LIN {X 0,Y 172.926,Z 518.236,A -85,B 0,C 180,E1 -23636.725,E2 -23636.725} C_VEL
LIN {X 0,Y 167.935,Z 527.248,A -85,B 0,C 180,E1 -23640.546,E2 -23640.546} C_VEL
LIN {X 0,Y 163.837,Z 534.508,A -85,B 0,C 180,E1 -23644.598,E2 -23644.598} C_VEL
LIN {X 0,Y 160.993,Z 539.589,A -85,B 0,C 180,E1 -23648.219,E2 -23648.219} C_VEL
LIN {X 0,Y 157.873,Z 544.852,A -85,B 0,C 180,E1 -23653.181,E2 -23653.181} C_VEL
LIN {X 0,Y 156.336,Z 547.79,A -85,B 0,C 180,E1 -23657.011,E2 -23657.011} C_VEL
LIN {X 0,Y 155.16,Z 550.483,A -85,B 0,C 180,E1 -23662.19,E2 -23662.19} C_VEL
LIN {X 0,Y 154.667,Z 551.827,A -85,B 0,C 180,E1 -23667.396,E2 -23667.396} C_VEL
LIN {X 0,Y 154.657,Z 551.936,A -85,B 0,C 180,E1 -23671.301,E2 -23671.301} C_VEL
LIN {X 0,Y 154.801,Z 551.368,A -85,B 0,C 180,E1 -23675.21,E2 -23675.21} C_VEL
LIN {X 0,Y 155.156,Z 550.552,A -85,B 0,C 180,E1 -23677.81,E2 -23677.81} C_VEL
LIN {X 0,Y 156.317,Z 547.899,A -85,B 0,C 180,E1 -23682.991,E2 -23682.991} C_VEL
LIN {X 0,Y 158.464,Z 543.823,A -85,B 0,C 180,E1 -23688.087,E2 -23688.087} C_VEL
LIN {X 0,Y 161.821,Z 538.19,A -85,B 0,C 180,E1 -23693.009,E2 -23693.009} C_VEL
LIN {X 0,Y 164.996,Z 532.618,A -85,B 0,C 180,E1 -23696.715,E2 -23696.715} C_VEL
LIN {X 0,Y 169.249,Z 525.15,A -85,B 0,C 180,E1 -23700.576,E2 -23700.576} C_VEL
LIN {X 0,Y 173.636,Z 517.128,A -85,B 0,C 180,E1 -23703.817,E2 -23703.817} C_VEL
LIN {X 0,Y 178.54,Z 507.453,A -85,B 0,C 180,E1 -23706.892,E2 -23706.892} C_VEL
LIN {X 0,Y 182.704,Z 498.37,A -85,B 0,C 180,E1 -23709.202,E2 -23709.202} C_VEL
LIN {X 0,Y 183.404,Z 491.819,A -85,B 0,C 180,E1 -23711.15,E2 -23711.15} C_VEL
LIN {X 0,Y 183.287,Z 481.855,A -85,B 0,C 180,E1 -23714.112,E2 -23714.112} C_VEL
LIN {X 0,Y 182.291,Z 472.749,A -85,B 0,C 180,E1 -23716.817,E2 -23716.817} C_VEL
LIN {X 0,Y 180.315,Z 464.485,A -85,B 0,C 180,E1 -23719.466,E2 -23719.466} C_VEL
LIN {X 0,Y 177.999,Z 458.041,A -85,B 0,C 180,E1 -23721.775,E2 -23721.775} C_VEL
LIN {X 0,Y 174.457,Z 449.919,A -85,B 0,C 180,E1 -23724.966,E2 -23724.966} C_VEL
LIN {X 0,Y 171.581,Z 444.63,A -85,B 0,C 180,E1 -23727.392,E2 -23727.392} C_VEL
LIN {X 0,Y 169.45,Z 440.565,A -85,B 0,C 180,E1 -23729.308,E2 -23729.308} C_VEL
LIN {X 0,Y 166.805,Z 436.801,A -85,B 0,C 180,E1 -23731.534,E2 -23731.534} C_VEL
LIN {X 0,Y 165.956,Z 434.977,A -85,B 0,C 180,E1 -23732.407,E2 -23732.407} C_VEL
LIN {X 0,Y 163.2,Z 432.01,A -85,B 0,C 180,E1 -23734.833,E2 -23734.833} C_VEL
LIN {X 0,Y 161.872,Z 429.259,A -85,B 0,C 180,E1 -23736.321,E2 -23736.321} C_VEL
LIN {X 0,Y 159.325,Z 427.59,A -85,B 0,C 180,E1 -23738.828,E2 -23738.828} C_VEL
LIN {X 0,Y 157.743,Z 424.933,A -85,B 0,C 180,E1 -23740.804,E2 -23740.804} C_VEL
LIN {X 0,Y 157.405,Z 423.504,A -85,B 0,C 180,E1 -23741.446,E2 -23741.446} C_VEL
LIN {X 0,Y 157.557,Z 423.483,A -85,B 0,C 180,E1 -23747.113,E2 -23747.113} C_VEL
LIN {X 0,Y 157.775,Z 423.457,A -85,B 0,C 180,E1 -23749.736,E2 -23749.736} C_VEL
LIN {X 0,Y 157.827,Z 423.452,A -85,B 0,C 180,E1 -23752.323,E2 -23752.323} C_VEL
LIN {X 0,Y 158.26,Z 423.396,A -85,B 0,C 180,E1 -23760,E2 -23760} C_VEL
LIN {X 0,Y 157.827,Z 423.449,A -85,B 0,C 180,E1 -23767.677,E2 -23767.677} C_VEL
LIN {X 0,Y 157.708,Z 423.466,A -85,B 0,C 180,E1 -23771.362,E2 -23771.362} C_VEL
LIN {X 0,Y 157.481,Z 423.493,A -85,B 0,C 180,E1 -23775.531,E2 -23775.531} C_VEL
LIN {X 0,Y 157.471,Z 423.801,A -85,B 0,C 180,E1 -23778.604,E2 -23778.604} C_VEL
LIN {X 0,Y 158.285,Z 426.09,A -85,B 0,C 180,E1 -23779.816,E2 -23779.816} C_VEL
LIN {X 0,Y 160.246,Z 428.772,A -85,B 0,C 180,E1 -23782.057,E2 -23782.057} C_VEL
LIN {X 0,Y 162.347,Z 430.594,A -85,B 0,C 180,E1 -23784.114,E2 -23784.114} C_VEL
LIN {X 0,Y 164.079,Z 434.137,A -85,B 0,C 180,E1 -23785.974,E2 -23785.974} C_VEL
LIN {X 0,Y 166.374,Z 436.806,A -85,B 0,C 180,E1 -23787.969,E2 -23787.969} C_VEL
LIN {X 0,Y 168.403,Z 440.705,A -85,B 0,C 180,E1 -23789.88,E2 -23789.88} C_VEL
LIN {X 0,Y 169.659,Z 442.431,A -85,B 0,C 180,E1 -23790.887,E2 -23790.887} C_VEL
LIN {X 0,Y 172.027,Z 446.791,A -85,B 0,C 180,E1 -23792.947,E2 -23792.947} C_VEL
LIN {X 0,Y 175.71,Z 454.541,A -85,B 0,C 180,E1 -23796.154,E2 -23796.154} C_VEL
LIN {X 0,Y 178.774,Z 462.124,A -85,B 0,C 180,E1 -23798.976,E2 -23798.976} C_VEL
LIN {X 0,Y 181.187,Z 470.196,A -85,B 0,C 180,E1 -23801.677,E2 -23801.677} C_VEL
LIN {X 0,Y 182.199,Z 476.723,A -85,B 0,C 180,E1 -23803.59,E2 -23803.59} C_VEL
LIN {X 0,Y 182.759,Z 485.981,A -85,B 0,C 180,E1 -23806.196,E2 -23806.196} C_VEL
LIN {X 0,Y 182.442,Z 495.967,A -85,B 0,C 180,E1 -23809.09,E2 -23809.09} C_VEL
LIN {X 0,Y 181.954,Z 500.895,A -85,B 0,C 180,E1 -23810.579,E2 -23810.579} C_VEL
LIN {X 0,Y 181.533,Z 502.814,A -85,B 0,C 180,E1 -23811.119,E2 -23811.119} C_VEL
LIN {X 0,Y 176.391,Z 513.568,A -85,B 0,C 180,E1 -23814.006,E2 -23814.006} C_VEL
LIN {X 0,Y 171.669,Z 522.688,A -85,B 0,C 180,E1 -23817.149,E2 -23817.149} C_VEL
LIN {X 0,Y 166.779,Z 531.405,A -85,B 0,C 180,E1 -23821.013,E2 -23821.013} C_VEL
LIN {X 0,Y 162.662,Z 538.52,A -85,B 0,C 180,E1 -23825.139,E2 -23825.139} C_VEL
LIN {X 0,Y 159.677,Z 544.066,A -85,B 0,C 180,E1 -23829.383,E2 -23829.383} C_VEL
LIN {X 0,Y 156.925,Z 548.946,A -85,B 0,C 180,E1 -23834.412,E2 -23834.412} C_VEL
LIN {X 0,Y 155.389,Z 552.34,A -85,B 0,C 180,E1 -23839.577,E2 -23839.577} C_VEL
LIN {X 0,Y 154.695,Z 554.346,A -85,B 0,C 180,E1 -23844.786,E2 -23844.786} C_VEL
LIN {X 0,Y 154.684,Z 555.005,A -85,B 0,C 180,E1 -23850,E2 -23850} C_VEL
LIN {X 0,Y 154.695,Z 554.325,A -85,B 0,C 180,E1 -23855.213,E2 -23855.213} C_VEL
LIN {X 0,Y 155.39,Z 552.301,A -85,B 0,C 180,E1 -23860.423,E2 -23860.423} C_VEL
LIN {X 0,Y 156.92,Z 548.885,A -85,B 0,C 180,E1 -23865.588,E2 -23865.588} C_VEL
LIN {X 0,Y 159.688,Z 543.979,A -85,B 0,C 180,E1 -23870.615,E2 -23870.615} C_VEL
LIN {X 0,Y 162.854,Z 538.174,A -85,B 0,C 180,E1 -23875.007,E2 -23875.007} C_VEL
LIN {X 0,Y 166.773,Z 531.27,A -85,B 0,C 180,E1 -23878.988,E2 -23878.988} C_VEL
LIN {X 0,Y 171.692,Z 522.522,A -85,B 0,C 180,E1 -23882.845,E2 -23882.845} C_VEL
LIN {X 0,Y 176.409,Z 513.368,A -85,B 0,C 180,E1 -23885.989,E2 -23885.989} C_VEL
LIN {X 0,Y 178.015,Z 510.091,A -85,B 0,C 180,E1 -23886.936,E2 -23886.936} C_VEL
LIN {X 0,Y 178.978,Z 507.362,A -85,B 0,C 180,E1 -23887.774,E2 -23887.774} C_VEL
LIN {X 0,Y 179.272,Z 503.359,A -85,B 0,C 180,E1 -23889.176,E2 -23889.176} C_VEL
LIN {X 0,Y 178.699,Z 499.6,A -85,B 0,C 180,E1 -23890.654,E2 -23890.654} C_VEL
LIN {X 0,Y 177.025,Z 491.821,A -85,B 0,C 180,E1 -23893.689,E2 -23893.689} C_VEL
LIN {X 0,Y 176.838,Z 488.942,A -85,B 0,C 180,E1 -23894.631,E2 -23894.631} C_VEL
LIN {X 0,Y 176.635,Z 479.607,A -85,B 0,C 180,E1 -23897.437,E2 -23897.437} C_VEL
LIN {X 0,Y 175.522,Z 472.284,A -85,B 0,C 180,E1 -23899.778,E2 -23899.778} C_VEL
LIN {X 0,Y 173.933,Z 466.481,A -85,B 0,C 180,E1 -23901.855,E2 -23901.855} C_VEL
LIN {X 0,Y 171.092,Z 458.845,A -85,B 0,C 180,E1 -23904.895,E2 -23904.895} C_VEL
LIN {X 0,Y 168.211,Z 452.209,A -85,B 0,C 180,E1 -23907.812,E2 -23907.812} C_VEL
LIN {X 0,Y 166.109,Z 447.895,A -85,B 0,C 180,E1 -23909.927,E2 -23909.927} C_VEL
LIN {X 0,Y 163.64,Z 443.734,A -85,B 0,C 180,E1 -23912.33,E2 -23912.33} C_VEL
LIN {X 0,Y 163.002,Z 442.254,A -85,B 0,C 180,E1 -23913.082,E2 -23913.082} C_VEL
LIN {X 0,Y 160.807,Z 439.375,A -85,B 0,C 180,E1 -23915.242,E2 -23915.242} C_VEL
LIN {X 0,Y 159.571,Z 436.565,A -85,B 0,C 180,E1 -23916.819,E2 -23916.819} C_VEL
LIN {X 0,Y 156.742,Z 433.546,A -85,B 0,C 180,E1 -23920.017,E2 -23920.017} C_VEL
LIN {X 0,Y 155.337,Z 430.302,A -85,B 0,C 180,E1 -23922.218,E2 -23922.218} C_VEL
LIN {X 0,Y 152.287,Z 428.264,A -85,B 0,C 180,E1 -23926.81,E2 -23926.81} C_VEL
LIN {X 0,Y 150.954,Z 425.405,A -85,B 0,C 180,E1 -23930.03,E2 -23930.03} C_VEL
LIN {X 0,Y 150.722,Z 424.337,A -85,B 0,C 180,E1 -23930.946,E2 -23930.946} C_VEL
LIN {X 0,Y 150.903,Z 424.313,A -85,B 0,C 180,E1 -23937.331,E2 -23937.331} C_VEL
LIN {X 0,Y 151.221,Z 424.272,A -85,B 0,C 180,E1 -23940,E2 -23940} C_VEL
LIN {X 0,Y 150.764,Z 424.33,A -85,B 0,C 180,E1 -23948.039,E2 -23948.039} C_VEL
LIN {X 0,Y 150.746,Z 424.431,A -85,B 0,C 180,E1 -23949.391,E2 -23949.391} C_VEL
LIN {X 0,Y 151.619,Z 427.253,A -85,B 0,C 180,E1 -23952.009,E2 -23952.009} C_VEL
LIN {X 0,Y 153.548,Z 429.386,A -85,B 0,C 180,E1 -23955.599,E2 -23955.599} C_VEL
LIN {X 0,Y 155.496,Z 430.531,A -85,B 0,C 180,E1 -23958.274,E2 -23958.274} C_VEL
LIN {X 0,Y 156.695,Z 433.412,A -85,B 0,C 180,E1 -23960.169,E2 -23960.169} C_VEL
LIN {X 0,Y 159.006,Z 435.579,A -85,B 0,C 180,E1 -23962.795,E2 -23962.795} C_VEL
LIN {X 0,Y 159.683,Z 436.232,A -85,B 0,C 180,E1 -23963.514,E2 -23963.514} C_VEL
LIN {X 0,Y 161.638,Z 439.756,A -85,B 0,C 180,E1 -23965.773,E2 -23965.773} C_VEL
LIN {X 0,Y 163.321,Z 441.724,A -85,B 0,C 180,E1 -23967.381,E2 -23967.381} C_VEL
LIN {X 0,Y 166.904,Z 448.442,A -85,B 0,C 180,E1 -23971.053,E2 -23971.053} C_VEL
LIN {X 0,Y 168.703,Z 451.832,A -85,B 0,C 180,E1 -23972.791,E2 -23972.791} C_VEL
LIN {X 0,Y 171.618,Z 458.27,A -85,B 0,C 180,E1 -23975.701,E2 -23975.701} C_VEL
LIN {X 0,Y 174.36,Z 465.65,A -85,B 0,C 180,E1 -23978.665,E2 -23978.665} C_VEL
LIN {X 0,Y 176.184,Z 472.574,A -85,B 0,C 180,E1 -23981.161,E2 -23981.161} C_VEL
LIN {X 0,Y 177.218,Z 479.908,A -85,B 0,C 180,E1 -23983.566,E2 -23983.566} C_VEL
LIN {X 0,Y 177.528,Z 489.397,A -85,B 0,C 180,E1 -23986.532,E2 -23986.532} C_VEL
LIN {X 0,Y 176.984,Z 497.901,A -85,B 0,C 180,E1 -23989.268,E2 -23989.268} C_VEL
LIN {X 0,Y 176.815,Z 499.083,A -85,B 0,C 180,E1 -23989.638,E2 -23989.638} C_VEL
LIN {X 0,Y 172.036,Z 508.857,A -85,B 0,C 180,E1 -23992.21,E2 -23992.21} C_VEL
LIN {X 0,Y 167.013,Z 518.308,A -85,B 0,C 180,E1 -23995.383,E2 -23995.383} C_VEL
LIN {X 0,Y 161.766,Z 527.319,A -85,B 0,C 180,E1 -23999.304,E2 -23999.304} C_VEL
LIN {X 0,Y 157.381,Z 534.579,A -85,B 0,C 180,E1 -24003.477,E2 -24003.477} C_VEL
LIN {X 0,Y 154.393,Z 539.66,A -85,B 0,C 180,E1 -24007.237,E2 -24007.237} C_VEL
LIN {X 0,Y 151.045,Z 544.923,A -85,B 0,C 180,E1 -24012.396,E2 -24012.396} C_VEL
LIN {X 0,Y 149.41,Z 547.859,A -85,B 0,C 180,E1 -24016.397,E2 -24016.397} C_VEL
LIN {X 0,Y 148.102,Z 550.552,A -85,B 0,C 180,E1 -24021.816,E2 -24021.816} C_VEL
LIN {X 0,Y 147.572,Z 551.896,A -85,B 0,C 180,E1 -24027.271,E2 -24027.271} C_VEL
LIN {X 0,Y 147.597,Z 552.049,A -85,B 0,C 180,E1 -24030.614,E2 -24030.614} C_VEL
LIN {X 0,Y 147.727,Z 551.437,A -85,B 0,C 180,E1 -24035.46,E2 -24035.46} C_VEL
LIN {X 0,Y 148.604,Z 549.466,A -85,B 0,C 180,E1 -24040.905,E2 -24040.905} C_VEL
LIN {X 0,Y 150.419,Z 546.114,A -85,B 0,C 180,E1 -24046.281,E2 -24046.281} C_VEL
LIN {X 0,Y 153.413,Z 541.278,A -85,B 0,C 180,E1 -24051.499,E2 -24051.499} C_VEL
LIN {X 0,Y 157.396,Z 534.805,A -85,B 0,C 180,E1 -24056.521,E2 -24056.521} C_VEL
LIN {X 0,Y 161.734,Z 527.596,A -85,B 0,C 180,E1 -24060.703,E2 -24060.703} C_VEL
LIN {X 0,Y 166.938,Z 518.674,A -85,B 0,C 180,E1 -24064.635,E2 -24064.635} C_VEL
LIN {X 0,Y 172.006,Z 509.298,A -85,B 0,C 180,E1 -24067.799,E2 -24067.799} C_VEL
LIN {X 0,Y 176.72,Z 499.621,A -85,B 0,C 180,E1 -24070.386,E2 -24070.386} C_VEL
LIN {X 0,Y 177.522,Z 492.221,A -85,B 0,C 180,E1 -24072.722,E2 -24072.722} C_VEL
LIN {X 0,Y 177.517,Z 482.496,A -85,B 0,C 180,E1 -24075.784,E2 -24075.784} C_VEL
LIN {X 0,Y 176.693,Z 474.887,A -85,B 0,C 180,E1 -24078.223,E2 -24078.223} C_VEL
LIN {X 0,Y 175.181,Z 468.219,A -85,B 0,C 180,E1 -24080.558,E2 -24080.558} C_VEL
LIN {X 0,Y 172.912,Z 461.554,A -85,B 0,C 180,E1 -24083.165,E2 -24083.165} C_VEL
LIN {X 0,Y 170.239,Z 454.885,A -85,B 0,C 180,E1 -24085.986,E2 -24085.986} C_VEL
LIN {X 0,Y 167.733,Z 449.906,A -85,B 0,C 180,E1 -24088.416,E2 -24088.416} C_VEL
LIN {X 0,Y 165.651,Z 445.799,A -85,B 0,C 180,E1 -24090.535,E2 -24090.535} C_VEL
LIN {X 0,Y 163.358,Z 441.764,A -85,B 0,C 180,E1 -24092.886,E2 -24092.886} C_VEL
LIN {X 0,Y 160.147,Z 437.275,A -85,B 0,C 180,E1 -24096.222,E2 -24096.222} C_VEL
LIN {X 0,Y 159.511,Z 435.836,A -85,B 0,C 180,E1 -24097.067,E2 -24097.067} C_VEL
LIN {X 0,Y 157.043,Z 433.825,A -85,B 0,C 180,E1 -24099.796,E2 -24099.796} C_VEL
LIN {X 0,Y 155.502,Z 430.56,A -85,B 0,C 180,E1 -24102.152,E2 -24102.152} C_VEL
LIN {X 0,Y 152.111,Z 427.998,A -85,B 0,C 180,E1 -24107.546,E2 -24107.546} C_VEL
LIN {X 0,Y 150.805,Z 424.729,A -85,B 0,C 180,E1 -24111.204,E2 -24111.204} C_VEL
LIN {X 0,Y 150.749,Z 424.33,A -85,B 0,C 180,E1 -24111.623,E2 -24111.623} C_VEL
LIN {X 0,Y 151.221,Z 424.273,A -85,B 0,C 180,E1 -24120,E2 -24120} C_VEL
LIN {X 0,Y 150.739,Z 424.365,A -85,B 0,C 180,E1 -24128.378,E2 -24128.378} C_VEL
LIN {X 0,Y 151.542,Z 426.956,A -85,B 0,C 180,E1 -24130.996,E2 -24130.996} C_VEL
LIN {X 0,Y 153.348,Z 429.262,A -85,B 0,C 180,E1 -24134.6,E2 -24134.6} C_VEL
LIN {X 0,Y 155.559,Z 430.611,A -85,B 0,C 180,E1 -24137.755,E2 -24137.755} C_VEL
LIN {X 0,Y 157.293,Z 434.31,A -85,B 0,C 180,E1 -24140.38,E2 -24140.38} C_VEL
LIN {X 0,Y 159.896,Z 437.055,A -85,B 0,C 180,E1 -24143.302,E2 -24143.302} C_VEL
LIN {X 0,Y 161.729,Z 440.76,A -85,B 0,C 180,E1 -24145.498,E2 -24145.498} C_VEL
LIN {X 0,Y 163.385,Z 442.899,A -85,B 0,C 180,E1 -24147.109,E2 -24147.109} C_VEL
LIN {X 0,Y 165.56,Z 447.084,A -85,B 0,C 180,E1 -24149.395,E2 -24149.395} C_VEL
LIN {X 0,Y 166.06,Z 447.7,A -85,B 0,C 180,E1 -24149.82,E2 -24149.82} C_VEL
LIN {X 0,Y 168.931,Z 453.785,A -85,B 0,C 180,E1 -24152.74,E2 -24152.74} C_VEL
LIN {X 0,Y 172.407,Z 461.832,A -85,B 0,C 180,E1 -24156.233,E2 -24156.233} C_VEL
LIN {X 0,Y 175.431,Z 471.484,A -85,B 0,C 180,E1 -24159.865,E2 -24159.865} C_VEL
LIN {X 0,Y 176.511,Z 477.442,A -85,B 0,C 180,E1 -24161.829,E2 -24161.829} C_VEL
LIN {X 0,Y 176.965,Z 486.961,A -85,B 0,C 180,E1 -24164.692,E2 -24164.692} C_VEL
LIN {X 0,Y 176.609,Z 495.895,A -85,B 0,C 180,E1 -24167.429,E2 -24167.429} C_VEL
LIN {X 0,Y 175.69,Z 503.255,A -85,B 0,C 180,E1 -24169.76,E2 -24169.76} C_VEL
LIN {X 0,Y 171.568,Z 511.821,A -85,B 0,C 180,E1 -24172.088,E2 -24172.088} C_VEL
LIN {X 0,Y 166.469,Z 521.245,A -85,B 0,C 180,E1 -24175.253,E2 -24175.253} C_VEL
LIN {X 0,Y 161.277,Z 530.22,A -85,B 0,C 180,E1 -24179.2,E2 -24179.2} C_VEL
LIN {X 0,Y 156.849,Z 537.475,A -85,B 0,C 180,E1 -24183.38,E2 -24183.38} C_VEL
LIN {X 0,Y 152.987,Z 543.998,A -85,B 0,C 180,E1 -24188.438,E2 -24188.438} C_VEL
LIN {X 0,Y 150.057,Z 548.877,A -85,B 0,C 180,E1 -24193.679,E2 -24193.679} C_VEL
LIN {X 0,Y 148.374,Z 552.271,A -85,B 0,C 180,E1 -24199.078,E2 -24199.078} C_VEL
LIN {X 0,Y 147.623,Z 554.277,A -85,B 0,C 180,E1 -24204.536,E2 -24204.536} C_VEL
LIN {X 0,Y 147.588,Z 554.936,A -85,B 0,C 180,E1 -24210,E2 -24210} C_VEL
LIN {X 0,Y 147.623,Z 554.255,A -85,B 0,C 180,E1 -24215.463,E2 -24215.463} C_VEL
LIN {X 0,Y 148.374,Z 552.231,A -85,B 0,C 180,E1 -24220.921,E2 -24220.921} C_VEL
LIN {X 0,Y 150.053,Z 548.815,A -85,B 0,C 180,E1 -24226.321,E2 -24226.321} C_VEL
LIN {X 0,Y 153.002,Z 543.908,A -85,B 0,C 180,E1 -24231.56,E2 -24231.56} C_VEL
LIN {X 0,Y 156.143,Z 538.54,A -85,B 0,C 180,E1 -24235.816,E2 -24235.816} C_VEL
LIN {X 0,Y 160.574,Z 531.199,A -85,B 0,C 180,E1 -24240.22,E2 -24240.22} C_VEL
LIN {X 0,Y 165.74,Z 522.451,A -85,B 0,C 180,E1 -24244.184,E2 -24244.184} C_VEL
LIN {X 0,Y 170.696,Z 513.296,A -85,B 0,C 180,E1 -24247.394,E2 -24247.394} C_VEL
LIN {X 0,Y 175.66,Z 503.055,A -85,B 0,C 180,E1 -24250.228,E2 -24250.228} C_VEL
LIN {X 0,Y 176.704,Z 493.056,A -85,B 0,C 180,E1 -24253.378,E2 -24253.378} C_VEL
LIN {X 0,Y 176.838,Z 488.942,A -85,B 0,C 180,E1 -24254.631,E2 -24254.631} C_VEL
LIN {X 0,Y 176.306,Z 484.941,A -85,B 0,C 180,E1 -24256.029,E2 -24256.029} C_VEL
LIN {X 0,Y 174.873,Z 481.493,A -85,B 0,C 180,E1 -24257.542,E2 -24257.542} C_VEL
LIN {X 0,Y 169.938,Z 473.071,A -85,B 0,C 180,E1 -24261.821,E2 -24261.821} C_VEL
LIN {X 0,Y 169.036,Z 470.649,A -85,B 0,C 180,E1 -24262.874,E2 -24262.874} C_VEL
LIN {X 0,Y 166.521,Z 463.123,A -85,B 0,C 180,E1 -24266.094,E2 -24266.094} C_VEL
LIN {X 0,Y 163.981,Z 456.991,A -85,B 0,C 180,E1 -24269.049,E2 -24269.049} C_VEL
LIN {X 0,Y 162.458,Z 453.39,A -85,B 0,C 180,E1 -24270.878,E2 -24270.878} C_VEL
LIN {X 0,Y 160.342,Z 449.38,A -85,B 0,C 180,E1 -24273.303,E2 -24273.303} C_VEL
LIN {X 0,Y 159.278,Z 447.608,A -85,B 0,C 180,E1 -24274.519,E2 -24274.519} C_VEL
LIN {X 0,Y 157.237,Z 443.663,A -85,B 0,C 180,E1 -24277.151,E2 -24277.151} C_VEL
LIN {X 0,Y 156.533,Z 442.51,A -85,B 0,C 180,E1 -24278.086,E2 -24278.086} C_VEL
LIN {X 0,Y 154.245,Z 439.526,A -85,B 0,C 180,E1 -24281.115,E2 -24281.115} C_VEL
LIN {X 0,Y 153.232,Z 436.998,A -85,B 0,C 180,E1 -24282.999,E2 -24282.999} C_VEL
LIN {X 0,Y 150.601,Z 434.94,A -85,B 0,C 180,E1 -24287.42,E2 -24287.42} C_VEL
LIN {X 0,Y 149.422,Z 432.001,A -85,B 0,C 180,E1 -24290.884,E2 -24290.884} C_VEL
LIN {X 0,Y 149.306,Z 431.322,A -85,B 0,C 180,E1 -24291.491,E2 -24291.491} C_VEL
LIN {X 0,Y 147.774,Z 430.484,A -85,B 0,C 180,E1 -24300,E2 -24300} C_VEL
LIN {X 0,Y 149.308,Z 431.378,A -85,B 0,C 180,E1 -24308.8,E2 -24308.8} C_VEL
LIN {X 0,Y 150.294,Z 434.547,A -85,B 0,C 180,E1 -24312.181,E2 -24312.181} C_VEL
LIN {X 0,Y 152.563,Z 436.717,A -85,B 0,C 180,E1 -24316.389,E2 -24316.389} C_VEL
LIN {X 0,Y 153.357,Z 437.198,A -85,B 0,C 180,E1 -24317.524,E2 -24317.524} C_VEL
LIN {X 0,Y 154.614,Z 440.165,A -85,B 0,C 180,E1 -24319.76,E2 -24319.76} C_VEL
LIN {X 0,Y 157.066,Z 442.636,A -85,B 0,C 180,E1 -24322.789,E2 -24322.789} C_VEL
LIN {X 0,Y 158.902,Z 446.104,A -85,B 0,C 180,E1 -24325.195,E2 -24325.195} C_VEL
LIN {X 0,Y 160.283,Z 448.011,A -85,B 0,C 180,E1 -24326.708,E2 -24326.708} C_VEL
LIN {X 0,Y 164.429,Z 456.285,A -85,B 0,C 180,E1 -24331.501,E2 -24331.501} C_VEL
LIN {X 0,Y 167.452,Z 463.802,A -85,B 0,C 180,E1 -24335.089,E2 -24335.089} C_VEL
LIN {X 0,Y 169.914,Z 471.524,A -85,B 0,C 180,E1 -24338.348,E2 -24338.348} C_VEL
LIN {X 0,Y 171.296,Z 478.694,A -85,B 0,C 180,E1 -24341.03,E2 -24341.03} C_VEL
LIN {X 0,Y 171.774,Z 486.393,A -85,B 0,C 180,E1 -24343.664,E2 -24343.664} C_VEL
LIN {X 0,Y 171.489,Z 494.96,A -85,B 0,C 180,E1 -24346.53,E2 -24346.53} C_VEL
LIN {X 0,Y 170.883,Z 500.342,A -85,B 0,C 180,E1 -24348.379,E2 -24348.379} C_VEL
LIN {X 0,Y 165.553,Z 510.633,A -85,B 0,C 180,E1 -24351.233,E2 -24351.233} C_VEL
LIN {X 0,Y 160.395,Z 519.773,A -85,B 0,C 180,E1 -24354.509,E2 -24354.509} C_VEL
LIN {X 0,Y 154.972,Z 528.503,A -85,B 0,C 180,E1 -24358.565,E2 -24358.565} C_VEL
LIN {X 0,Y 151.012,Z 534.65,A -85,B 0,C 180,E1 -24362.265,E2 -24362.265} C_VEL
LIN {X 0,Y 146.849,Z 541.168,A -85,B 0,C 180,E1 -24367.489,E2 -24367.489} C_VEL
LIN {X 0,Y 143.61,Z 546.053,A -85,B 0,C 180,E1 -24372.925,E2 -24372.925} C_VEL
LIN {X 0,Y 141.638,Z 549.448,A -85,B 0,C 180,E1 -24378.552,E2 -24378.552} C_VEL
LIN {X 0,Y 140.655,Z 551.459,A -85,B 0,C 180,E1 -24384.265,E2 -24384.265} C_VEL
LIN {X 0,Y 140.524,Z 552.141,A -85,B 0,C 180,E1 -24390,E2 -24390} C_VEL
LIN {X 0,Y 140.654,Z 551.505,A -85,B 0,C 180,E1 -24395.736,E2 -24395.736} C_VEL
LIN {X 0,Y 141.626,Z 549.535,A -85,B 0,C 180,E1 -24401.449,E2 -24401.449} C_VEL
LIN {X 0,Y 143.572,Z 546.182,A -85,B 0,C 180,E1 -24407.08,E2 -24407.08} C_VEL
LIN {X 0,Y 146.812,Z 541.346,A -85,B 0,C 180,E1 -24412.518,E2 -24412.518} C_VEL
LIN {X 0,Y 151.013,Z 534.873,A -85,B 0,C 180,E1 -24417.736,E2 -24417.736} C_VEL
LIN {X 0,Y 155.647,Z 527.664,A -85,B 0,C 180,E1 -24422.043,E2 -24422.043} C_VEL
LIN {X 0,Y 161.146,Z 518.741,A -85,B 0,C 180,E1 -24426.07,E2 -24426.07} C_VEL
LIN {X 0,Y 166.447,Z 509.364,A -85,B 0,C 180,E1 -24429.298,E2 -24429.298} C_VEL
LIN {X 0,Y 170.824,Z 500.796,A -85,B 0,C 180,E1 -24431.649,E2 -24431.649} C_VEL
LIN {X 0,Y 171.71,Z 492.378,A -85,B 0,C 180,E1 -24434.51,E2 -24434.51} C_VEL
LIN {X 0,Y 171.821,Z 483.724,A -85,B 0,C 180,E1 -24437.414,E2 -24437.414} C_VEL
LIN {X 0,Y 171.166,Z 477.13,A -85,B 0,C 180,E1 -24439.707,E2 -24439.707} C_VEL
LIN {X 0,Y 169.694,Z 470.441,A -85,B 0,C 180,E1 -24442.271,E2 -24442.271} C_VEL
LIN {X 0,Y 166.768,Z 461.825,A -85,B 0,C 180,E1 -24446.035,E2 -24446.035} C_VEL
LIN {X 0,Y 164.149,Z 455.711,A -85,B 0,C 180,E1 -24449.084,E2 -24449.084} C_VEL
LIN {X 0,Y 162.061,Z 451.341,A -85,B 0,C 180,E1 -24451.508,E2 -24451.508} C_VEL
LIN {X 0,Y 160.059,Z 447.326,A -85,B 0,C 180,E1 -24453.954,E2 -24453.954} C_VEL
LIN {X 0,Y 157.548,Z 443.745,A -85,B 0,C 180,E1 -24456.851,E2 -24456.851} C_VEL
LIN {X 0,Y 157.052,Z 442.433,A -85,B 0,C 180,E1 -24457.643,E2 -24457.643} C_VEL
LIN {X 0,Y 154.75,Z 440.25,A -85,B 0,C 180,E1 -24460.489,E2 -24460.489} C_VEL
LIN {X 0,Y 153.336,Z 437.052,A -85,B 0,C 180,E1 -24463.011,E2 -24463.011} C_VEL
LIN {X 0,Y 150.754,Z 435.125,A -85,B 0,C 180,E1 -24467.412,E2 -24467.412} C_VEL
LIN {X 0,Y 149.474,Z 432.114,A -85,B 0,C 180,E1 -24471.305,E2 -24471.305} C_VEL
LIN {X 0,Y 149.186,Z 431.244,A -85,B 0,C 180,E1 -24472.556,E2 -24472.556} C_VEL
LIN {X 0,Y 148.077,Z 430.62,A -85,B 0,C 180,E1 -24480,E2 -24480} C_VEL
LIN {X 0,Y 149.372,Z 431.501,A -85,B 0,C 180,E1 -24487.944,E2 -24487.944} C_VEL
LIN {X 0,Y 150.738,Z 435.101,A -85,B 0,C 180,E1 -24492.34,E2 -24492.34} C_VEL
LIN {X 0,Y 153.53,Z 437.424,A -85,B 0,C 180,E1 -24497.117,E2 -24497.117} C_VEL
LIN {X 0,Y 155.202,Z 441.021,A -85,B 0,C 180,E1 -24499.958,E2 -24499.958} C_VEL
LIN {X 0,Y 157.232,Z 443.385,A -85,B 0,C 180,E1 -24502.503,E2 -24502.503} C_VEL
LIN {X 0,Y 159.202,Z 447.421,A -85,B 0,C 180,E1 -24505.144,E2 -24505.144} C_VEL
LIN {X 0,Y 160.082,Z 448.427,A -85,B 0,C 180,E1 -24506.042,E2 -24506.042} C_VEL
LIN {X 0,Y 162.035,Z 452.746,A -85,B 0,C 180,E1 -24508.496,E2 -24508.496} C_VEL
LIN {X 0,Y 164.531,Z 457.871,A -85,B 0,C 180,E1 -24511.316,E2 -24511.316} C_VEL
LIN {X 0,Y 167.846,Z 466.528,A -85,B 0,C 180,E1 -24515.306,E2 -24515.306} C_VEL
LIN {X 0,Y 170.378,Z 475.691,A -85,B 0,C 180,E1 -24518.98,E2 -24518.98} C_VEL
LIN {X 0,Y 171.169,Z 481.679,A -85,B 0,C 180,E1 -24521.067,E2 -24521.067} C_VEL
LIN {X 0,Y 171.222,Z 490.355,A -85,B 0,C 180,E1 -24523.859,E2 -24523.859} C_VEL
LIN {X 0,Y 170.5,Z 499.166,A -85,B 0,C 180,E1 -24526.743,E2 -24526.743} C_VEL
LIN {X 0,Y 169.709,Z 504.349,A -85,B 0,C 180,E1 -24528.502,E2 -24528.502} C_VEL
LIN {X 0,Y 165.068,Z 513.435,A -85,B 0,C 180,E1 -24531.097,E2 -24531.097} C_VEL
LIN {X 0,Y 159.846,Z 522.554,A -85,B 0,C 180,E1 -24534.368,E2 -24534.368} C_VEL
LIN {X 0,Y 154.473,Z 531.27,A -85,B 0,C 180,E1 -24538.452,E2 -24538.452} C_VEL
LIN {X 0,Y 150.515,Z 537.407,A -85,B 0,C 180,E1 -24542.164,E2 -24542.164} C_VEL
LIN {X 0,Y 147.291,Z 542.495,A -85,B 0,C 180,E1 -24546.072,E2 -24546.072} C_VEL
LIN {X 0,Y 143.907,Z 547.742,A -85,B 0,C 180,E1 -24551.491,E2 -24551.491} C_VEL
LIN {X 0,Y 142.163,Z 550.684,A -85,B 0,C 180,E1 -24555.689,E2 -24555.689} C_VEL
LIN {X 0,Y 140.844,Z 553.375,A -85,B 0,C 180,E1 -24561.39,E2 -24561.39} C_VEL
LIN {X 0,Y 140.42,Z 554.705,A -85,B 0,C 180,E1 -24567.131,E2 -24567.131} C_VEL
LIN {X 0,Y 140.484,Z 554.867,A -85,B 0,C 180,E1 -24570,E2 -24570} C_VEL
LIN {X 0,Y 140.547,Z 554.186,A -85,B 0,C 180,E1 -24575.739,E2 -24575.739} C_VEL
LIN {X 0,Y 141.382,Z 552.162,A -85,B 0,C 180,E1 -24581.469,E2 -24581.469} C_VEL
LIN {X 0,Y 143.211,Z 548.745,A -85,B 0,C 180,E1 -24587.124,E2 -24587.124} C_VEL
LIN {X 0,Y 146.367,Z 543.838,A -85,B 0,C 180,E1 -24592.59,E2 -24592.59} C_VEL
LIN {X 0,Y 149.484,Z 538.884,A -85,B 0,C 180,E1 -24596.711,E2 -24596.711} C_VEL
LIN {X 0,Y 153.753,Z 532.246,A -85,B 0,C 180,E1 -24600.946,E2 -24600.946} C_VEL
LIN {X 0,Y 159.073,Z 523.736,A -85,B 0,C 180,E1 -24605.054,E2 -24605.054} C_VEL
LIN {X 0,Y 164.185,Z 514.854,A -85,B 0,C 180,E1 -24608.365,E2 -24608.365} C_VEL
LIN {X 0,Y 168.863,Z 506.049,A -85,B 0,C 180,E1 -24610.958,E2 -24610.958} C_VEL
LIN {X 0,Y 169.684,Z 504.094,A -85,B 0,C 180,E1 -24611.505,E2 -24611.505} C_VEL
LIN {X 0,Y 170.883,Z 494.42,A -85,B 0,C 180,E1 -24614.742,E2 -24614.742} C_VEL
LIN {X 0,Y 171.196,Z 485.454,A -85,B 0,C 180,E1 -24617.641,E2 -24617.641} C_VEL
LIN {X 0,Y 170.881,Z 479.361,A -85,B 0,C 180,E1 -24619.627,E2 -24619.627} C_VEL
LIN {X 0,Y 169.776,Z 473.177,A -85,B 0,C 180,E1 -24621.861,E2 -24621.861} C_VEL
LIN {X 0,Y 169.036,Z 470.649,A -85,B 0,C 180,E1 -24622.874,E2 -24622.874} C_VEL
LIN {X 0,Y 167.515,Z 467.436,A -85,B 0,C 180,E1 -24624.473,E2 -24624.473} C_VEL
LIN {X 0,Y 165.379,Z 465.053,A -85,B 0,C 180,E1 -24626.195,E2 -24626.195} C_VEL
LIN {X 0,Y 159.311,Z 459.832,A -85,B 0,C 180,E1 -24631.121,E2 -24631.121} C_VEL
LIN {X 0,Y 158.193,Z 458.108,A -85,B 0,C 180,E1 -24632.37,E2 -24632.37} C_VEL
LIN {X 0,Y 156.551,Z 454.204,A -85,B 0,C 180,E1 -24634.756,E2 -24634.756} C_VEL
LIN {X 0,Y 154.691,Z 450.898,A -85,B 0,C 180,E1 -24637.283,E2 -24637.283} C_VEL
LIN {X 0,Y 153.953,Z 448.998,A -85,B 0,C 180,E1 -24638.58,E2 -24638.58} C_VEL
LIN {X 0,Y 151.711,Z 445.764,A -85,B 0,C 180,E1 -24641.953,E2 -24641.953} C_VEL
LIN {X 0,Y 151.079,Z 443.746,A -85,B 0,C 180,E1 -24643.446,E2 -24643.446} C_VEL
LIN {X 0,Y 148.68,Z 441.662,A -85,B 0,C 180,E1 -24647.892,E2 -24647.892} C_VEL
LIN {X 0,Y 147.667,Z 438.63,A -85,B 0,C 180,E1 -24651.594,E2 -24651.594} C_VEL
LIN {X 0,Y 147.463,Z 438.141,A -85,B 0,C 180,E1 -24652.469,E2 -24652.469} C_VEL
LIN {X 0,Y 146.312,Z 437.42,A -85,B 0,C 180,E1 -24660,E2 -24660} C_VEL
LIN {X 0,Y 147.595,Z 438.404,A -85,B 0,C 180,E1 -24668.385,E2 -24668.385} C_VEL
LIN {X 0,Y 148.41,Z 441.314,A -85,B 0,C 180,E1 -24671.784,E2 -24671.784} C_VEL
LIN {X 0,Y 150.848,Z 443.631,A -85,B 0,C 180,E1 -24676.581,E2 -24676.581} C_VEL
LIN {X 0,Y 151.966,Z 446.314,A -85,B 0,C 180,E1 -24678.889,E2 -24678.889} C_VEL
LIN {X 0,Y 153.749,Z 448.428,A -85,B 0,C 180,E1 -24681.45,E2 -24681.45} C_VEL
LIN {X 0,Y 156.462,Z 453.045,A -85,B 0,C 180,E1 -24685.26,E2 -24685.26} C_VEL
LIN {X 0,Y 159.905,Z 460.458,A -85,B 0,C 180,E1 -24689.934,E2 -24689.934} C_VEL
LIN {X 0,Y 162.452,Z 467.173,A -85,B 0,C 180,E1 -24693.477,E2 -24693.477} C_VEL
LIN {X 0,Y 164.535,Z 474.143,A -85,B 0,C 180,E1 -24696.727,E2 -24696.727} C_VEL
LIN {X 0,Y 165.78,Z 480.837,A -85,B 0,C 180,E1 -24699.487,E2 -24699.487} C_VEL
LIN {X 0,Y 166.148,Z 488.148,A -85,B 0,C 180,E1 -24702.183,E2 -24702.183} C_VEL
LIN {X 0,Y 165.538,Z 497.486,A -85,B 0,C 180,E1 -24705.533,E2 -24705.533} C_VEL
LIN {X 0,Y 164.967,Z 501.582,A -85,B 0,C 180,E1 -24707.028,E2 -24707.028} C_VEL
LIN {X 0,Y 160.06,Z 510.704,A -85,B 0,C 180,E1 -24709.636,E2 -24709.636} C_VEL
LIN {X 0,Y 154.635,Z 519.845,A -85,B 0,C 180,E1 -24712.973,E2 -24712.973} C_VEL
LIN {X 0,Y 148.931,Z 528.574,A -85,B 0,C 180,E1 -24717.134,E2 -24717.134} C_VEL
LIN {X 0,Y 144.716,Z 534.721,A -85,B 0,C 180,E1 -24720.946,E2 -24720.946} C_VEL
LIN {X 0,Y 140.301,Z 541.238,A -85,B 0,C 180,E1 -24726.376,E2 -24726.376} C_VEL
LIN {X 0,Y 136.793,Z 546.123,A -85,B 0,C 180,E1 -24732.046,E2 -24732.046} C_VEL
LIN {X 0,Y 134.681,Z 549.518,A -85,B 0,C 180,E1 -24737.952,E2 -24737.952} C_VEL
LIN {X 0,Y 133.581,Z 551.529,A -85,B 0,C 180,E1 -24743.96,E2 -24743.96} C_VEL
LIN {X 0,Y 133.449,Z 552.209,A -85,B 0,C 180,E1 -24750,E2 -24750} C_VEL
LIN {X 0,Y 133.58,Z 551.574,A -85,B 0,C 180,E1 -24756.04,E2 -24756.04} C_VEL
LIN {X 0,Y 134.039,Z 550.757,A -85,B 0,C 180,E1 -24759.05,E2 -24759.05} C_VEL
LIN {X 0,Y 135.564,Z 548.105,A -85,B 0,C 180,E1 -24765.024,E2 -24765.024} C_VEL
LIN {X 0,Y 138.328,Z 544.027,A -85,B 0,C 180,E1 -24770.834,E2 -24770.834} C_VEL
LIN {X 0,Y 141.291,Z 539.991,A -85,B 0,C 180,E1 -24775.012,E2 -24775.012} C_VEL
LIN {X 0,Y 144.717,Z 534.941,A -85,B 0,C 180,E1 -24779.055,E2 -24779.055} C_VEL
LIN {X 0,Y 149.664,Z 527.731,A -85,B 0,C 180,E1 -24783.488,E2 -24783.488} C_VEL
LIN {X 0,Y 155.462,Z 518.807,A -85,B 0,C 180,E1 -24787.612,E2 -24787.612} C_VEL
LIN {X 0,Y 161.016,Z 509.43,A -85,B 0,C 180,E1 -24790.899,E2 -24790.899} C_VEL
LIN {X 0,Y 164.914,Z 502.053,A -85,B 0,C 180,E1 -24792.99,E2 -24792.99} C_VEL
LIN {X 0,Y 165.917,Z 494.792,A -85,B 0,C 180,E1 -24795.63,E2 -24795.63} C_VEL
LIN {X 0,Y 166.253,Z 487.398,A -85,B 0,C 180,E1 -24798.257,E2 -24798.257} C_VEL
LIN {X 0,Y 165.751,Z 479.934,A -85,B 0,C 180,E1 -24801.057,E2 -24801.057} C_VEL
LIN {X 0,Y 164.282,Z 472.899,A -85,B 0,C 180,E1 -24804.043,E2 -24804.043} C_VEL
LIN {X 0,Y 161.619,Z 464.663,A -85,B 0,C 180,E1 -24808.018,E2 -24808.018} C_VEL
LIN {X 0,Y 158.867,Z 457.713,A -85,B 0,C 180,E1 -24811.854,E2 -24811.854} C_VEL
LIN {X 0,Y 156.752,Z 453.238,A -85,B 0,C 180,E1 -24814.79,E2 -24814.79} C_VEL
LIN {X 0,Y 154.037,Z 448.628,A -85,B 0,C 180,E1 -24818.592,E2 -24818.592} C_VEL
LIN {X 0,Y 151.681,Z 445.628,A -85,B 0,C 180,E1 -24822.123,E2 -24822.123} C_VEL
LIN {X 0,Y 150.939,Z 443.683,A -85,B 0,C 180,E1 -24823.777,E2 -24823.777} C_VEL
LIN {X 0,Y 148.545,Z 441.456,A -85,B 0,C 180,E1 -24828.573,E2 -24828.573} C_VEL
LIN {X 0,Y 147.66,Z 438.32,A -85,B 0,C 180,E1 -24832.479,E2 -24832.479} C_VEL
LIN {X 0,Y 146.607,Z 437.572,A -85,B 0,C 180,E1 -24840,E2 -24840} C_VEL
LIN {X 0,Y 147.677,Z 438.316,A -85,B 0,C 180,E1 -24847.348,E2 -24847.348} C_VEL
LIN {X 0,Y 148.845,Z 441.829,A -85,B 0,C 180,E1 -24851.921,E2 -24851.921} C_VEL
LIN {X 0,Y 151.233,Z 443.999,A -85,B 0,C 180,E1 -24856.45,E2 -24856.45} C_VEL
LIN {X 0,Y 152.778,Z 447.574,A -85,B 0,C 180,E1 -24859.482,E2 -24859.482} C_VEL
LIN {X 0,Y 154.167,Z 449.173,A -85,B 0,C 180,E1 -24861.389,E2 -24861.389} C_VEL
LIN {X 0,Y 155.738,Z 452.889,A -85,B 0,C 180,E1 -24863.963,E2 -24863.963} C_VEL
LIN {X 0,Y 156.758,Z 454.36,A -85,B 0,C 180,E1 -24865.209,E2 -24865.209} C_VEL
LIN {X 0,Y 159.426,Z 460.711,A -85,B 0,C 180,E1 -24869.007,E2 -24869.007} C_VEL
LIN {X 0,Y 162.175,Z 467.906,A -85,B 0,C 180,E1 -24872.799,E2 -24872.799} C_VEL
LIN {X 0,Y 164.187,Z 474.842,A -85,B 0,C 180,E1 -24875.98,E2 -24875.98} C_VEL
LIN {X 0,Y 165.394,Z 480.67,A -85,B 0,C 180,E1 -24878.4,E2 -24878.4} C_VEL
LIN {X 0,Y 165.763,Z 486.923,A -85,B 0,C 180,E1 -24880.67,E2 -24880.67} C_VEL
LIN {X 0,Y 165.278,Z 495.749,A -85,B 0,C 180,E1 -24883.707,E2 -24883.707} C_VEL
LIN {X 0,Y 164.013,Z 504.371,A -85,B 0,C 180,E1 -24886.757,E2 -24886.757} C_VEL
LIN {X 0,Y 163.001,Z 507.311,A -85,B 0,C 180,E1 -24887.691,E2 -24887.691} C_VEL
LIN {X 0,Y 156.751,Z 518.138,A -85,B 0,C 180,E1 -24891.119,E2 -24891.119} C_VEL
LIN {X 0,Y 151.576,Z 526.457,A -85,B 0,C 180,E1 -24894.579,E2 -24894.579} C_VEL
LIN {X 0,Y 146.24,Z 534.411,A -85,B 0,C 180,E1 -24898.894,E2 -24898.894} C_VEL
LIN {X 0,Y 141.822,Z 540.816,A -85,B 0,C 180,E1 -24903.513,E2 -24903.513} C_VEL
LIN {X 0,Y 137.974,Z 546.496,A -85,B 0,C 180,E1 -24909.111,E2 -24909.111} C_VEL
LIN {X 0,Y 135.269,Z 550.616,A -85,B 0,C 180,E1 -24914.943,E2 -24914.943} C_VEL
LIN {X 0,Y 133.817,Z 553.307,A -85,B 0,C 180,E1 -24920.935,E2 -24920.935} C_VEL
LIN {X 0,Y 133.326,Z 554.636,A -85,B 0,C 180,E1 -24926.978,E2 -24926.978} C_VEL
LIN {X 0,Y 133.391,Z 554.798,A -85,B 0,C 180,E1 -24930,E2 -24930} C_VEL
LIN {X 0,Y 133.464,Z 554.117,A -85,B 0,C 180,E1 -24936.045,E2 -24936.045} C_VEL
LIN {X 0,Y 134.414,Z 552.092,A -85,B 0,C 180,E1 -24942.072,E2 -24942.072} C_VEL
LIN {X 0,Y 136.401,Z 548.675,A -85,B 0,C 180,E1 -24948.008,E2 -24948.008} C_VEL
LIN {X 0,Y 139.791,Z 543.767,A -85,B 0,C 180,E1 -24953.716,E2 -24953.716} C_VEL
LIN {X 0,Y 144.26,Z 537.221,A -85,B 0,C 180,E1 -24959.155,E2 -24959.155} C_VEL
LIN {X 0,Y 149.189,Z 529.939,A -85,B 0,C 180,E1 -24963.608,E2 -24963.608} C_VEL
LIN {X 0,Y 154.962,Z 520.916,A -85,B 0,C 180,E1 -24967.753,E2 -24967.753} C_VEL
LIN {X 0,Y 160.599,Z 511.453,A -85,B 0,C 180,E1 -24971.027,E2 -24971.027} C_VEL
LIN {X 0,Y 163.465,Z 506.057,A -85,B 0,C 180,E1 -24972.587,E2 -24972.587} C_VEL
LIN {X 0,Y 164.966,Z 497.724,A -85,B 0,C 180,E1 -24975.528,E2 -24975.528} C_VEL
LIN {X 0,Y 165.568,Z 489.249,A -85,B 0,C 180,E1 -24978.454,E2 -24978.454} C_VEL
LIN {X 0,Y 165.563,Z 483.471,A -85,B 0,C 180,E1 -24980.451,E2 -24980.451} C_VEL
LIN {X 0,Y 164.907,Z 478.175,A -85,B 0,C 180,E1 -24982.474,E2 -24982.474} C_VEL
LIN {X 0,Y 162.89,Z 470.374,A -85,B 0,C 180,E1 -24985.883,E2 -24985.883} C_VEL
LIN {X 0,Y 159.959,Z 462.174,A -85,B 0,C 180,E1 -24990.025,E2 -24990.025} C_VEL
LIN {X 0,Y 158.803,Z 459.099,A -85,B 0,C 180,E1 -24991.664,E2 -24991.664} C_VEL
LIN {X 0,Y 158.193,Z 458.108,A -85,B 0,C 180,E1 -24992.37,E2 -24992.37} C_VEL
LIN {X 0,Y 156.993,Z 456.746,A -85,B 0,C 180,E1 -24993.643,E2 -24993.643} C_VEL
LIN {X 0,Y 154.424,Z 456.021,A -85,B 0,C 180,E1 -24995.886,E2 -24995.886} C_VEL
LIN {X 0,Y 151.435,Z 455.495,A -85,B 0,C 180,E1 -24998.718,E2 -24998.718} C_VEL
LIN {X 0,Y 150.692,Z 454.884,A -85,B 0,C 180,E1 -24999.675,E2 -24999.675} C_VEL
LIN {X 0,Y 149.225,Z 452.61,A -85,B 0,C 180,E1 -25002.174,E2 -25002.174} C_VEL
LIN {X 0,Y 148.686,Z 451.03,A -85,B 0,C 180,E1 -25003.525,E2 -25003.525} C_VEL
LIN {X 0,Y 145.887,Z 446.812,A -85,B 0,C 180,E1 -25010.468,E2 -25010.468} C_VEL
LIN {X 0,Y 145.628,Z 445.139,A -85,B 0,C 180,E1 -25012.374,E2 -25012.374} C_VEL
LIN {X 0,Y 144.524,Z 444.286,A -85,B 0,C 180,E1 -25020,E2 -25020} C_VEL
LIN {X 0,Y 145.578,Z 445.19,A -85,B 0,C 180,E1 -25027.891,E2 -25027.891} C_VEL
LIN {X 0,Y 146.145,Z 447.786,A -85,B 0,C 180,E1 -25031.091,E2 -25031.091} C_VEL
LIN {X 0,Y 148.497,Z 450.699,A -85,B 0,C 180,E1 -25036.497,E2 -25036.497} C_VEL
LIN {X 0,Y 149.735,Z 453.471,A -85,B 0,C 180,E1 -25039.181,E2 -25039.181} C_VEL
LIN {X 0,Y 151.352,Z 455.77,A -85,B 0,C 180,E1 -25041.807,E2 -25041.807} C_VEL
LIN {X 0,Y 152.99,Z 458.831,A -85,B 0,C 180,E1 -25044.421,E2 -25044.421} C_VEL
LIN {X 0,Y 155.827,Z 465.681,A -85,B 0,C 180,E1 -25049.002,E2 -25049.002} C_VEL
LIN {X 0,Y 158.166,Z 472.816,A -85,B 0,C 180,E1 -25052.979,E2 -25052.979} C_VEL
LIN {X 0,Y 159.82,Z 479.65,A -85,B 0,C 180,E1 -25056.336,E2 -25056.336} C_VEL
LIN {X 0,Y 160.603,Z 486.752,A -85,B 0,C 180,E1 -25059.383,E2 -25059.383} C_VEL
LIN {X 0,Y 160.329,Z 494.123,A -85,B 0,C 180,E1 -25062.209,E2 -25062.209} C_VEL
LIN {X 0,Y 159.354,Z 501.662,A -85,B 0,C 180,E1 -25065.118,E2 -25065.118} C_VEL
LIN {X 0,Y 159.129,Z 502.881,A -85,B 0,C 180,E1 -25065.597,E2 -25065.597} C_VEL
LIN {X 0,Y 154.715,Z 510.776,A -85,B 0,C 180,E1 -25067.931,E2 -25067.931} C_VEL
LIN {X 0,Y 148.998,Z 519.916,A -85,B 0,C 180,E1 -25071.319,E2 -25071.319} C_VEL
LIN {X 0,Y 143.005,Z 528.645,A -85,B 0,C 180,E1 -25075.586,E2 -25075.586} C_VEL
LIN {X 0,Y 137.632,Z 536.032,A -85,B 0,C 180,E1 -25080.458,E2 -25080.458} C_VEL
LIN {X 0,Y 133.807,Z 541.308,A -85,B 0,C 180,E1 -25085.154,E2 -25085.154} C_VEL
LIN {X 0,Y 130.017,Z 546.194,A -85,B 0,C 180,E1 -25091.076,E2 -25091.076} C_VEL
LIN {X 0,Y 127.715,Z 549.588,A -85,B 0,C 180,E1 -25097.284,E2 -25097.284} C_VEL
LIN {X 0,Y 126.532,Z 551.598,A -85,B 0,C 180,E1 -25103.622,E2 -25103.622} C_VEL
LIN {X 0,Y 126.36,Z 552.278,A -85,B 0,C 180,E1 -25110,E2 -25110} C_VEL
LIN {X 0,Y 126.532,Z 551.643,A -85,B 0,C 180,E1 -25116.378,E2 -25116.378} C_VEL
LIN {X 0,Y 127.681,Z 549.672,A -85,B 0,C 180,E1 -25122.72,E2 -25122.72} C_VEL
LIN {X 0,Y 129.987,Z 546.319,A -85,B 0,C 180,E1 -25128.93,E2 -25128.93} C_VEL
LIN {X 0,Y 133.755,Z 541.482,A -85,B 0,C 180,E1 -25134.857,E2 -25134.857} C_VEL
LIN {X 0,Y 138.189,Z 535.443,A -85,B 0,C 180,E1 -25140.164,E2 -25140.164} C_VEL
LIN {X 0,Y 142.951,Z 528.912,A -85,B 0,C 180,E1 -25144.429,E2 -25144.429} C_VEL
LIN {X 0,Y 148.948,Z 520.24,A -85,B 0,C 180,E1 -25148.697,E2 -25148.697} C_VEL
LIN {X 0,Y 154.685,Z 511.163,A -85,B 0,C 180,E1 -25152.079,E2 -25152.079} C_VEL
LIN {X 0,Y 159.11,Z 503.233,A -85,B 0,C 180,E1 -25154.461,E2 -25154.461} C_VEL
LIN {X 0,Y 160.129,Z 497.01,A -85,B 0,C 180,E1 -25156.857,E2 -25156.857} C_VEL
LIN {X 0,Y 160.721,Z 489.259,A -85,B 0,C 180,E1 -25159.836,E2 -25159.836} C_VEL
LIN {X 0,Y 160.468,Z 483.481,A -85,B 0,C 180,E1 -25162.181,E2 -25162.181} C_VEL
LIN {X 0,Y 159.397,Z 477.203,A -85,B 0,C 180,E1 -25165.027,E2 -25165.027} C_VEL
LIN {X 0,Y 157.193,Z 469.422,A -85,B 0,C 180,E1 -25169.058,E2 -25169.058} C_VEL
LIN {X 0,Y 154.83,Z 462.827,A -85,B 0,C 180,E1 -25173.004,E2 -25173.004} C_VEL
LIN {X 0,Y 153.26,Z 459.052,A -85,B 0,C 180,E1 -25175.625,E2 -25175.625} C_VEL
LIN {X 0,Y 150.866,Z 454.62,A -85,B 0,C 180,E1 -25179.55,E2 -25179.55} C_VEL
LIN {X 0,Y 149.261,Z 452.599,A -85,B 0,C 180,E1 -25182.178,E2 -25182.178} C_VEL
LIN {X 0,Y 148.711,Z 451.125,A -85,B 0,C 180,E1 -25183.527,E2 -25183.527} C_VEL
LIN {X 0,Y 146.369,Z 448.173,A -85,B 0,C 180,E1 -25188.927,E2 -25188.927} C_VEL
LIN {X 0,Y 145.668,Z 445.014,A -85,B 0,C 180,E1 -25193.072,E2 -25193.072} C_VEL
LIN {X 0,Y 144.817,Z 444.424,A -85,B 0,C 180,E1 -25200,E2 -25200} C_VEL
LIN {X 0,Y 145.712,Z 445.153,A -85,B 0,C 180,E1 -25206.925,E2 -25206.925} C_VEL
LIN {X 0,Y 146.504,Z 448.227,A -85,B 0,C 180,E1 -25211.063,E2 -25211.063} C_VEL
LIN {X 0,Y 148.876,Z 451.335,A -85,B 0,C 180,E1 -25216.454,E2 -25216.454} C_VEL
LIN {X 0,Y 150.15,Z 454.108,A -85,B 0,C 180,E1 -25219.126,E2 -25219.126} C_VEL
LIN {X 0,Y 150.998,Z 455.168,A -85,B 0,C 180,E1 -25220.431,E2 -25220.431} C_VEL
LIN {X 0,Y 153.263,Z 460.142,A -85,B 0,C 180,E1 -25224.375,E2 -25224.375} C_VEL
LIN {X 0,Y 155.814,Z 467.05,A -85,B 0,C 180,E1 -25228.711,E2 -25228.711} C_VEL
LIN {X 0,Y 158.267,Z 474.858,A -85,B 0,C 180,E1 -25232.954,E2 -25232.954} C_VEL
LIN {X 0,Y 159.853,Z 482.337,A -85,B 0,C 180,E1 -25236.471,E2 -25236.471} C_VEL
LIN {X 0,Y 160.313,Z 487.654,A -85,B 0,C 180,E1 -25238.661,E2 -25238.661} C_VEL
LIN {X 0,Y 159.8,Z 495.675,A -85,B 0,C 180,E1 -25241.612,E2 -25241.612} C_VEL
LIN {X 0,Y 158.86,Z 502.276,A -85,B 0,C 180,E1 -25244.054,E2 -25244.054} C_VEL
LIN {X 0,Y 157.748,Z 507.253,A -85,B 0,C 180,E1 -25245.934,E2 -25245.934} C_VEL
LIN {X 0,Y 151.286,Z 518.071,A -85,B 0,C 180,E1 -25249.43,E2 -25249.43} C_VEL
LIN {X 0,Y 145.828,Z 526.39,A -85,B 0,C 180,E1 -25252.956,E2 -25252.956} C_VEL
LIN {X 0,Y 140.172,Z 534.343,A -85,B 0,C 180,E1 -25257.385,E2 -25257.385} C_VEL
LIN {X 0,Y 135.446,Z 540.748,A -85,B 0,C 180,E1 -25262.161,E2 -25262.161} C_VEL
LIN {X 0,Y 131.336,Z 546.427,A -85,B 0,C 180,E1 -25268.001,E2 -25268.001} C_VEL
LIN {X 0,Y 128.387,Z 550.547,A -85,B 0,C 180,E1 -25274.115,E2 -25274.115} C_VEL
LIN {X 0,Y 126.786,Z 553.238,A -85,B 0,C 180,E1 -25280.427,E2 -25280.427} C_VEL
LIN {X 0,Y 126.242,Z 554.567,A -85,B 0,C 180,E1 -25286.808,E2 -25286.808} C_VEL
LIN {X 0,Y 126.307,Z 554.73,A -85,B 0,C 180,E1 -25290,E2 -25290} C_VEL
LIN {X 0,Y 126.407,Z 554.048,A -85,B 0,C 180,E1 -25296.384,E2 -25296.384} C_VEL
LIN {X 0,Y 127.441,Z 552.022,A -85,B 0,C 180,E1 -25302.743,E2 -25302.743} C_VEL
LIN {X 0,Y 129.632,Z 548.605,A -85,B 0,C 180,E1 -25308.983,E2 -25308.983} C_VEL
LIN {X 0,Y 133.282,Z 543.697,A -85,B 0,C 180,E1 -25314.951,E2 -25314.951} C_VEL
LIN {X 0,Y 136.764,Z 538.925,A -85,B 0,C 180,E1 -25319.257,E2 -25319.257} C_VEL
LIN {X 0,Y 141.706,Z 532.104,A -85,B 0,C 180,E1 -25323.914,E2 -25323.914} C_VEL
LIN {X 0,Y 147.596,Z 523.593,A -85,B 0,C 180,E1 -25328.244,E2 -25328.244} C_VEL
LIN {X 0,Y 153.268,Z 514.711,A -85,B 0,C 180,E1 -25331.673,E2 -25331.673} C_VEL
LIN {X 0,Y 157.643,Z 507.181,A -85,B 0,C 180,E1 -25334.016,E2 -25334.016} C_VEL
LIN {X 0,Y 159.105,Z 499.982,A -85,B 0,C 180,E1 -25336.709,E2 -25336.709} C_VEL
LIN {X 0,Y 160.082,Z 491.039,A -85,B 0,C 180,E1 -25340.01,E2 -25340.01} C_VEL
LIN {X 0,Y 160.104,Z 485.276,A -85,B 0,C 180,E1 -25342.198,E2 -25342.198} C_VEL
LIN {X 0,Y 159.357,Z 479.871,A -85,B 0,C 180,E1 -25344.534,E2 -25344.534} C_VEL
LIN {X 0,Y 157.645,Z 472.956,A -85,B 0,C 180,E1 -25347.891,E2 -25347.891} C_VEL
LIN {X 0,Y 154.911,Z 464.575,A -85,B 0,C 180,E1 -25352.544,E2 -25352.544} C_VEL
LIN {X 0,Y 153.067,Z 459.967,A -85,B 0,C 180,E1 -25355.592,E2 -25355.592} C_VEL
LIN {X 0,Y 150.692,Z 454.884,A -85,B 0,C 180,E1 -25359.675,E2 -25359.675} C_VEL
LIN {X 0,Y 149.152,Z 453.71,A -85,B 0,C 180,E1 -25361.806,E2 -25361.806} C_VEL
LIN {X 0,Y 146.421,Z 453.442,A -85,B 0,C 180,E1 -25365.493,E2 -25365.493} C_VEL
LIN {X 0,Y 143.855,Z 453.402,A -85,B 0,C 180,E1 -25370.109,E2 -25370.109} C_VEL
LIN {X 0,Y 143.389,Z 452.884,A -85,B 0,C 180,E1 -25371.672,E2 -25371.672} C_VEL
LIN {X 0,Y 142.971,Z 451.623,A -85,B 0,C 180,E1 -25374.358,E2 -25374.358} C_VEL
LIN {X 0,Y 142.414,Z 451.07,A -85,B 0,C 180,E1 -25380,E2 -25380} C_VEL
LIN {X 0,Y 142.879,Z 451.591,A -85,B 0,C 180,E1 -25385.646,E2 -25385.646} C_VEL
LIN {X 0,Y 143.314,Z 452.792,A -85,B 0,C 180,E1 -25388.46,E2 -25388.46} C_VEL
LIN {X 0,Y 144.631,Z 455.909,A -85,B 0,C 180,E1 -25393.628,E2 -25393.628} C_VEL
LIN {X 0,Y 145.922,Z 458.042,A -85,B 0,C 180,E1 -25396.797,E2 -25396.797} C_VEL
LIN {X 0,Y 148.071,Z 461.836,A -85,B 0,C 180,E1 -25401.158,E2 -25401.158} C_VEL
LIN {X 0,Y 150.043,Z 466.314,A -85,B 0,C 180,E1 -25404.933,E2 -25404.933} C_VEL
LIN {X 0,Y 152.293,Z 472.941,A -85,B 0,C 180,E1 -25409.401,E2 -25409.401} C_VEL
LIN {X 0,Y 153.978,Z 479.62,A -85,B 0,C 180,E1 -25413.211,E2 -25413.211} C_VEL
LIN {X 0,Y 154.998,Z 486.483,A -85,B 0,C 180,E1 -25416.633,E2 -25416.633} C_VEL
LIN {X 0,Y 155.104,Z 491.32,A -85,B 0,C 180,E1 -25418.767,E2 -25418.767} C_VEL
LIN {X 0,Y 154.462,Z 498.081,A -85,B 0,C 180,E1 -25421.547,E2 -25421.547} C_VEL
LIN {X 0,Y 153.389,Z 504.181,A -85,B 0,C 180,E1 -25424.055,E2 -25424.055} C_VEL
LIN {X 0,Y 149.523,Z 510.847,A -85,B 0,C 180,E1 -25426.109,E2 -25426.109} C_VEL
LIN {X 0,Y 143.511,Z 519.987,A -85,B 0,C 180,E1 -25429.543,E2 -25429.543} C_VEL
LIN {X 0,Y 137.184,Z 528.716,A -85,B 0,C 180,E1 -25433.904,E2 -25433.904} C_VEL
LIN {X 0,Y 131.85,Z 535.598,A -85,B 0,C 180,E1 -25438.523,E2 -25438.523} C_VEL
LIN {X 0,Y 127.363,Z 541.379,A -85,B 0,C 180,E1 -25443.804,E2 -25443.804} C_VEL
LIN {X 0,Y 123.288,Z 546.264,A -85,B 0,C 180,E1 -25450,E2 -25450} C_VEL
LIN {X 0,Y 120.778,Z 549.657,A -85,B 0,C 180,E1 -25456.541,E2 -25456.541} C_VEL
LIN {X 0,Y 119.473,Z 551.667,A -85,B 0,C 180,E1 -25463.244,E2 -25463.244} C_VEL
LIN {X 0,Y 119.279,Z 552.347,A -85,B 0,C 180,E1 -25470,E2 -25470} C_VEL
LIN {X 0,Y 119.472,Z 551.711,A -85,B 0,C 180,E1 -25476.757,E2 -25476.757} C_VEL
LIN {X 0,Y 120.749,Z 549.74,A -85,B 0,C 180,E1 -25483.463,E2 -25483.463} C_VEL
LIN {X 0,Y 123.26,Z 546.388,A -85,B 0,C 180,E1 -25490.006,E2 -25490.006} C_VEL
LIN {X 0,Y 127.314,Z 541.55,A -85,B 0,C 180,E1 -25496.207,E2 -25496.207} C_VEL
LIN {X 0,Y 132.431,Z 535.077,A -85,B 0,C 180,E1 -25502.053,E2 -25502.053} C_VEL
LIN {X 0,Y 138.001,Z 527.865,A -85,B 0,C 180,E1 -25506.755,E2 -25506.755} C_VEL
LIN {X 0,Y 144.451,Z 518.941,A -85,B 0,C 180,E1 -25511.058,E2 -25511.058} C_VEL
LIN {X 0,Y 150.561,Z 509.562,A -85,B 0,C 180,E1 -25514.442,E2 -25514.442} C_VEL
LIN {X 0,Y 153.395,Z 504.606,A -85,B 0,C 180,E1 -25515.958,E2 -25515.958} C_VEL
LIN {X 0,Y 154.992,Z 495.327,A -85,B 0,C 180,E1 -25519.749,E2 -25519.749} C_VEL
LIN {X 0,Y 155.219,Z 488.013,A -85,B 0,C 180,E1 -25522.86,E2 -25522.86} C_VEL
LIN {X 0,Y 154.386,Z 481.341,A -85,B 0,C 180,E1 -25526.106,E2 -25526.106} C_VEL
LIN {X 0,Y 152.927,Z 474.928,A -85,B 0,C 180,E1 -25529.634,E2 -25529.634} C_VEL
LIN {X 0,Y 150.948,Z 468.43,A -85,B 0,C 180,E1 -25533.748,E2 -25533.748} C_VEL
LIN {X 0,Y 149.587,Z 464.771,A -85,B 0,C 180,E1 -25536.462,E2 -25536.462} C_VEL
LIN {X 0,Y 147.497,Z 460.541,A -85,B 0,C 180,E1 -25540.516,E2 -25540.516} C_VEL
LIN {X 0,Y 145.056,Z 456.374,A -85,B 0,C 180,E1 -25545.98,E2 -25545.98} C_VEL
LIN {X 0,Y 144.061,Z 455.006,A -85,B 0,C 180,E1 -25548.747,E2 -25548.747} C_VEL
LIN {X 0,Y 143.19,Z 451.684,A -85,B 0,C 180,E1 -25554.366,E2 -25554.366} C_VEL
LIN {X 0,Y 142.7,Z 451.207,A -85,B 0,C 180,E1 -25560,E2 -25560} C_VEL
LIN {X 0,Y 143.261,Z 451.715,A -85,B 0,C 180,E1 -25565.63,E2 -25565.63} C_VEL
LIN {X 0,Y 145.88,Z 457.467,A -85,B 0,C 180,E1 -25575.519,E2 -25575.519} C_VEL
LIN {X 0,Y 147.64,Z 461.039,A -85,B 0,C 180,E1 -25579.464,E2 -25579.464} C_VEL
LIN {X 0,Y 149.885,Z 466.86,A -85,B 0,C 180,E1 -25584.222,E2 -25584.222} C_VEL
LIN {X 0,Y 151.985,Z 473.379,A -85,B 0,C 180,E1 -25588.527,E2 -25588.527} C_VEL
LIN {X 0,Y 153.659,Z 480.05,A -85,B 0,C 180,E1 -25592.299,E2 -25592.299} C_VEL
LIN {X 0,Y 154.684,Z 486.228,A -85,B 0,C 180,E1 -25595.401,E2 -25595.401} C_VEL
LIN {X 0,Y 154.905,Z 491.183,A -85,B 0,C 180,E1 -25597.592,E2 -25597.592} C_VEL
LIN {X 0,Y 153.862,Z 499.814,A -85,B 0,C 180,E1 -25600.995,E2 -25600.995} C_VEL
LIN {X 0,Y 152.439,Z 506.743,A -85,B 0,C 180,E1 -25603.753,E2 -25603.753} C_VEL
LIN {X 0,Y 151.45,Z 509.379,A -85,B 0,C 180,E1 -25604.745,E2 -25604.745} C_VEL
LIN {X 0,Y 144.926,Z 519.492,A -85,B 0,C 180,E1 -25608.18,E2 -25608.18} C_VEL
LIN {X 0,Y 139.283,Z 527.555,A -85,B 0,C 180,E1 -25611.821,E2 -25611.821} C_VEL
LIN {X 0,Y 133.449,Z 535.285,A -85,B 0,C 180,E1 -25616.428,E2 -25616.428} C_VEL
LIN {X 0,Y 129.135,Z 540.679,A -85,B 0,C 180,E1 -25620.671,E2 -25620.671} C_VEL
LIN {X 0,Y 124.754,Z 546.359,A -85,B 0,C 180,E1 -25626.774,E2 -25626.774} C_VEL
LIN {X 0,Y 121.521,Z 550.478,A -85,B 0,C 180,E1 -25633.191,E2 -25633.191} C_VEL
LIN {X 0,Y 119.755,Z 553.169,A -85,B 0,C 180,E1 -25639.859,E2 -25639.859} C_VEL
LIN {X 0,Y 119.15,Z 554.499,A -85,B 0,C 180,E1 -25646.618,E2 -25646.618} C_VEL
LIN {X 0,Y 119.226,Z 554.661,A -85,B 0,C 180,E1 -25650,E2 -25650} C_VEL
LIN {X 0,Y 119.328,Z 553.978,A -85,B 0,C 180,E1 -25656.764,E2 -25656.764} C_VEL
LIN {X 0,Y 120.498,Z 551.952,A -85,B 0,C 180,E1 -25663.491,E2 -25663.491} C_VEL
LIN {X 0,Y 122.912,Z 548.535,A -85,B 0,C 180,E1 -25670.064,E2 -25670.064} C_VEL
LIN {X 0,Y 126.846,Z 543.626,A -85,B 0,C 180,E1 -25676.311,E2 -25676.311} C_VEL
LIN {X 0,Y 130.55,Z 538.894,A -85,B 0,C 180,E1 -25680.756,E2 -25680.756} C_VEL
LIN {X 0,Y 135.835,Z 532.033,A -85,B 0,C 180,E1 -25685.596,E2 -25685.596} C_VEL
LIN {X 0,Y 142.049,Z 523.521,A -85,B 0,C 180,E1 -25690.029,E2 -25690.029} C_VEL
LIN {X 0,Y 148.018,Z 514.639,A -85,B 0,C 180,E1 -25693.509,E2 -25693.509} C_VEL
LIN {X 0,Y 151.875,Z 508.282,A -85,B 0,C 180,E1 -25695.541,E2 -25695.541} C_VEL
LIN {X 0,Y 153.602,Z 500.627,A -85,B 0,C 180,E1 -25698.599,E2 -25698.599} C_VEL
LIN {X 0,Y 154.722,Z 492.043,A -85,B 0,C 180,E1 -25701.967,E2 -25701.967} C_VEL
LIN {X 0,Y 154.607,Z 485.987,A -85,B 0,C 180,E1 -25704.579,E2 -25704.579} C_VEL
LIN {X 0,Y 153.477,Z 479.501,A -85,B 0,C 180,E1 -25707.846,E2 -25707.846} C_VEL
LIN {X 0,Y 151.369,Z 471.742,A -85,B 0,C 180,E1 -25712.336,E2 -25712.336} C_VEL
LIN {X 0,Y 149.395,Z 465.655,A -85,B 0,C 180,E1 -25716.43,E2 -25716.43} C_VEL
LIN {X 0,Y 147.424,Z 460.878,A -85,B 0,C 180,E1 -25720.506,E2 -25720.506} C_VEL
LIN {X 0,Y 145.022,Z 456.288,A -85,B 0,C 180,E1 -25725.977,E2 -25725.977} C_VEL
LIN {X 0,Y 143.389,Z 452.884,A -85,B 0,C 180,E1 -25731.672,E2 -25731.672} C_VEL
LIN {X 0,Y 142.98,Z 452.543,A -85,B 0,C 180,E1 -25733.229,E2 -25733.229} C_VEL
LIN {X 0,Y 142.465,Z 452.832,A -85,B 0,C 180,E1 -25734.793,E2 -25734.793} C_VEL
LIN {X 0,Y 141.332,Z 454.578,A -85,B 0,C 180,E1 -25737.897,E2 -25737.897} C_VEL
LIN {X 0,Y 140.139,Z 457.686,A -85,B 0,C 180,E1 -25742.665,E2 -25742.665} C_VEL
LIN {X 0,Y 140.178,Z 458.161,A -85,B 0,C 180,E1 -25744.304,E2 -25744.304} C_VEL
LIN {X 0,Y 140.4,Z 458.35,A -85,B 0,C 180,E1 -25745.746,E2 -25745.746} C_VEL
LIN {X 0,Y 140.738,Z 459.674,A -85,B 0,C 180,E1 -25748.616,E2 -25748.616} C_VEL
LIN {X 0,Y 142.579,Z 463.916,A -85,B 0,C 180,E1 -25755.73,E2 -25755.73} C_VEL
LIN {X 0,Y 144.294,Z 467.305,A -85,B 0,C 180,E1 -25759.935,E2 -25759.935} C_VEL
LIN {X 0,Y 145.966,Z 471.459,A -85,B 0,C 180,E1 -25763.821,E2 -25763.821} C_VEL
LIN {X 0,Y 147.81,Z 477.75,A -85,B 0,C 180,E1 -25768.391,E2 -25768.391} C_VEL
LIN {X 0,Y 149.221,Z 485.05,A -85,B 0,C 180,E1 -25772.793,E2 -25772.793} C_VEL
LIN {X 0,Y 149.731,Z 490.888,A -85,B 0,C 180,E1 -25775.872,E2 -25775.872} C_VEL
LIN {X 0,Y 149.448,Z 496.275,A -85,B 0,C 180,E1 -25778.372,E2 -25778.372} C_VEL
LIN {X 0,Y 148.149,Z 503.686,A -85,B 0,C 180,E1 -25781.617,E2 -25781.617} C_VEL
LIN {X 0,Y 147.739,Z 505.523,A -85,B 0,C 180,E1 -25782.417,E2 -25782.417} C_VEL
LIN {X 0,Y 145.609,Z 509.216,A -85,B 0,C 180,E1 -25783.615,E2 -25783.615} C_VEL
LIN {X 0,Y 139.193,Z 518.666,A -85,B 0,C 180,E1 -25787.029,E2 -25787.029} C_VEL
LIN {X 0,Y 132.414,Z 527.673,A -85,B 0,C 180,E1 -25791.418,E2 -25791.418} C_VEL
LIN {X 0,Y 126.438,Z 534.933,A -85,B 0,C 180,E1 -25796.231,E2 -25796.231} C_VEL
LIN {X 0,Y 120.983,Z 541.449,A -85,B 0,C 180,E1 -25802.308,E2 -25802.308} C_VEL
LIN {X 0,Y 116.607,Z 546.334,A -85,B 0,C 180,E1 -25808.8,E2 -25808.8} C_VEL
LIN {X 0,Y 113.873,Z 549.727,A -85,B 0,C 180,E1 -25815.708,E2 -25815.708} C_VEL
LIN {X 0,Y 112.437,Z 551.736,A -85,B 0,C 180,E1 -25822.819,E2 -25822.819} C_VEL
LIN {X 0,Y 112.199,Z 552.415,A -85,B 0,C 180,E1 -25830,E2 -25830} C_VEL
LIN {X 0,Y 112.434,Z 551.78,A -85,B 0,C 180,E1 -25837.182,E2 -25837.182} C_VEL
LIN {X 0,Y 113.819,Z 549.809,A -85,B 0,C 180,E1 -25844.3,E2 -25844.3} C_VEL
LIN {X 0,Y 116.581,Z 546.456,A -85,B 0,C 180,E1 -25851.205,E2 -25851.205} C_VEL
LIN {X 0,Y 120.936,Z 541.618,A -85,B 0,C 180,E1 -25857.705,E2 -25857.705} C_VEL
LIN {X 0,Y 125.371,Z 536.39,A -85,B 0,C 180,E1 -25862.768,E2 -25862.768} C_VEL
LIN {X 0,Y 131.443,Z 529.046,A -85,B 0,C 180,E1 -25867.944,E2 -25867.944} C_VEL
LIN {X 0,Y 138.146,Z 520.373,A -85,B 0,C 180,E1 -25872.383,E2 -25872.383} C_VEL
LIN {X 0,Y 144.458,Z 511.296,A -85,B 0,C 180,E1 -25875.857,E2 -25875.857} C_VEL
LIN {X 0,Y 147.75,Z 505.902,A -85,B 0,C 180,E1 -25877.598,E2 -25877.598} C_VEL
LIN {X 0,Y 149.383,Z 497.766,A -85,B 0,C 180,E1 -25881.149,E2 -25881.149} C_VEL
LIN {X 0,Y 149.848,Z 491.419,A -85,B 0,C 180,E1 -25884.065,E2 -25884.065} C_VEL
LIN {X 0,Y 149.538,Z 486.739,A -85,B 0,C 180,E1 -25886.481,E2 -25886.481} C_VEL
LIN {X 0,Y 148.337,Z 479.744,A -85,B 0,C 180,E1 -25890.581,E2 -25890.581} C_VEL
LIN {X 0,Y 146.895,Z 473.917,A -85,B 0,C 180,E1 -25894.495,E2 -25894.495} C_VEL
LIN {X 0,Y 145.738,Z 470.377,A -85,B 0,C 180,E1 -25897.307,E2 -25897.307} C_VEL
LIN {X 0,Y 143.942,Z 466.337,A -85,B 0,C 180,E1 -25901.496,E2 -25901.496} C_VEL
LIN {X 0,Y 142.36,Z 463.146,A -85,B 0,C 180,E1 -25905.709,E2 -25905.709} C_VEL
LIN {X 0,Y 140.684,Z 458.499,A -85,B 0,C 180,E1 -25914.266,E2 -25914.266} C_VEL
LIN {X 0,Y 140.268,Z 457.881,A -85,B 0,C 180,E1 -25920,E2 -25920} C_VEL
LIN {X 0,Y 140.749,Z 458.574,A -85,B 0,C 180,E1 -25925.731,E2 -25925.731} C_VEL
LIN {X 0,Y 142.556,Z 463.309,A -85,B 0,C 180,E1 -25934.27,E2 -25934.27} C_VEL
LIN {X 0,Y 144.082,Z 466.813,A -85,B 0,C 180,E1 -25938.485,E2 -25938.485} C_VEL
LIN {X 0,Y 145.728,Z 471.401,A -85,B 0,C 180,E1 -25942.694,E2 -25942.694} C_VEL
LIN {X 0,Y 147.582,Z 478.467,A -85,B 0,C 180,E1 -25947.665,E2 -25947.665} C_VEL
LIN {X 0,Y 148.944,Z 485.496,A -85,B 0,C 180,E1 -25951.859,E2 -25951.859} C_VEL
LIN {X 0,Y 149.546,Z 492.009,A -85,B 0,C 180,E1 -25955.277,E2 -25955.277} C_VEL
LIN {X 0,Y 148.989,Z 497.83,A -85,B 0,C 180,E1 -25957.823,E2 -25957.823} C_VEL
LIN {X 0,Y 147.46,Z 505.462,A -85,B 0,C 180,E1 -25961.057,E2 -25961.057} C_VEL
LIN {X 0,Y 146.304,Z 509.447,A -85,B 0,C 180,E1 -25962.751,E2 -25962.751} C_VEL
LIN {X 0,Y 140.77,Z 517.938,A -85,B 0,C 180,E1 -25965.656,E2 -25965.656} C_VEL
LIN {X 0,Y 134.736,Z 526.255,A -85,B 0,C 180,E1 -25969.306,E2 -25969.306} C_VEL
LIN {X 0,Y 128.386,Z 534.208,A -85,B 0,C 180,E1 -25973.951,E2 -25973.951} C_VEL
LIN {X 0,Y 122.957,Z 540.611,A -85,B 0,C 180,E1 -25979.041,E2 -25979.041} C_VEL
LIN {X 0,Y 118.234,Z 546.291,A -85,B 0,C 180,E1 -25985.412,E2 -25985.412} C_VEL
LIN {X 0,Y 114.693,Z 550.41,A -85,B 0,C 180,E1 -25992.158,E2 -25992.158} C_VEL
LIN {X 0,Y 112.751,Z 553.101,A -85,B 0,C 180,E1 -25999.222,E2 -25999.222} C_VEL
LIN {X 0,Y 112.058,Z 554.43,A -85,B 0,C 180,E1 -26006.404,E2 -26006.404} C_VEL
LIN {X 0,Y 112.133,Z 554.592,A -85,B 0,C 180,E1 -26010,E2 -26010} C_VEL
LIN {X 0,Y 112.264,Z 553.909,A -85,B 0,C 180,E1 -26017.192,E2 -26017.192} C_VEL
LIN {X 0,Y 113.585,Z 551.883,A -85,B 0,C 180,E1 -26024.329,E2 -26024.329} C_VEL
LIN {X 0,Y 116.248,Z 548.465,A -85,B 0,C 180,E1 -26031.268,E2 -26031.268} C_VEL
LIN {X 0,Y 120.49,Z 543.556,A -85,B 0,C 180,E1 -26037.815,E2 -26037.815} C_VEL
LIN {X 0,Y 124.463,Z 538.824,A -85,B 0,C 180,E1 -26042.439,E2 -26042.439} C_VEL
LIN {X 0,Y 130.102,Z 531.962,A -85,B 0,C 180,E1 -26047.424,E2 -26047.424} C_VEL
LIN {X 0,Y 136.652,Z 523.45,A -85,B 0,C 180,E1 -26051.958,E2 -26051.958} C_VEL
LIN {X 0,Y 142.94,Z 514.567,A -85,B 0,C 180,E1 -26055.473,E2 -26055.473} C_VEL
LIN {X 0,Y 146.2,Z 509.388,A -85,B 0,C 180,E1 -26057.182,E2 -26057.182} C_VEL
LIN {X 0,Y 148.234,Z 501.29,A -85,B 0,C 180,E1 -26060.638,E2 -26060.638} C_VEL
LIN {X 0,Y 149.238,Z 495.177,A -85,B 0,C 180,E1 -26063.184,E2 -26063.184} C_VEL
LIN {X 0,Y 149.371,Z 489.912,A -85,B 0,C 180,E1 -26065.625,E2 -26065.625} C_VEL
LIN {X 0,Y 148.431,Z 482.997,A -85,B 0,C 180,E1 -26069.403,E2 -26069.403} C_VEL
LIN {X 0,Y 146.903,Z 476.092,A -85,B 0,C 180,E1 -26073.735,E2 -26073.735} C_VEL
LIN {X 0,Y 145.547,Z 471.223,A -85,B 0,C 180,E1 -26077.276,E2 -26077.276} C_VEL
LIN {X 0,Y 143.883,Z 466.621,A -85,B 0,C 180,E1 -26081.489,E2 -26081.489} C_VEL
LIN {X 0,Y 142.345,Z 463.113,A -85,B 0,C 180,E1 -26085.708,E2 -26085.708} C_VEL
LIN {X 0,Y 140.493,Z 458.41,A -85,B 0,C 180,E1 -26094.258,E2 -26094.258} C_VEL
LIN {X 0,Y 139.993,Z 457.732,A -85,B 0,C 180,E1 -26100,E2 -26100} C_VEL
LIN {X 0,Y 140.178,Z 458.161,A -85,B 0,C 180,E1 -26104.304,E2 -26104.304} C_VEL
LIN {X 0,Y 140.278,Z 458.765,A -85,B 0,C 180,E1 -26105.883,E2 -26105.883} C_VEL
LIN {X 0,Y 140.121,Z 460.791,A -85,B 0,C 180,E1 -26108.148,E2 -26108.148} C_VEL
LIN {X 0,Y 139.215,Z 469.431,A -85,B 0,C 180,E1 -26114.677,E2 -26114.677} C_VEL
LIN {X 0,Y 139.501,Z 470.839,A -85,B 0,C 180,E1 -26116.226,E2 -26116.226} C_VEL
LIN {X 0,Y 140.979,Z 474.219,A -85,B 0,C 180,E1 -26120.424,E2 -26120.424} C_VEL
LIN {X 0,Y 141.993,Z 477.258,A -85,B 0,C 180,E1 -26123.326,E2 -26123.326} C_VEL
LIN {X 0,Y 143.141,Z 482.239,A -85,B 0,C 180,E1 -26127.18,E2 -26127.18} C_VEL
LIN {X 0,Y 144.004,Z 487.738,A -85,B 0,C 180,E1 -26130.827,E2 -26130.827} C_VEL
LIN {X 0,Y 144.392,Z 493.434,A -85,B 0,C 180,E1 -26134.163,E2 -26134.163} C_VEL
LIN {X 0,Y 144.081,Z 497.998,A -85,B 0,C 180,E1 -26136.507,E2 -26136.507} C_VEL
LIN {X 0,Y 142.628,Z 505.126,A -85,B 0,C 180,E1 -26139.835,E2 -26139.835} C_VEL
LIN {X 0,Y 141.614,Z 508.073,A -85,B 0,C 180,E1 -26141.159,E2 -26141.159} C_VEL
LIN {X 0,Y 135.121,Z 517.255,A -85,B 0,C 180,E1 -26144.343,E2 -26144.343} C_VEL
LIN {X 0,Y 128.878,Z 525.337,A -85,B 0,C 180,E1 -26148.086,E2 -26148.086} C_VEL
LIN {X 0,Y 122.281,Z 533.076,A -85,B 0,C 180,E1 -26152.881,E2 -26152.881} C_VEL
LIN {X 0,Y 117.494,Z 538.477,A -85,B 0,C 180,E1 -26157.429,E2 -26157.429} C_VEL
LIN {X 0,Y 112.186,Z 544.156,A -85,B 0,C 180,E1 -26163.991,E2 -26163.991} C_VEL
LIN {X 0,Y 108.288,Z 548.279,A -85,B 0,C 180,E1 -26171.065,E2 -26171.065} C_VEL
LIN {X 0,Y 106.036,Z 550.969,A -85,B 0,C 180,E1 -26178.531,E2 -26178.531} C_VEL
LIN {X 0,Y 105.052,Z 552.31,A -85,B 0,C 180,E1 -26186.164,E2 -26186.164} C_VEL
LIN {X 0,Y 105.106,Z 552.484,A -85,B 0,C 180,E1 -26190,E2 -26190} C_VEL
LIN {X 0,Y 105.373,Z 551.849,A -85,B 0,C 180,E1 -26197.666,E2 -26197.666} C_VEL
LIN {X 0,Y 106.929,Z 549.877,A -85,B 0,C 180,E1 -26205.243,E2 -26205.243} C_VEL
LIN {X 0,Y 109.961,Z 546.524,A -85,B 0,C 180,E1 -26212.55,E2 -26212.55} C_VEL
LIN {X 0,Y 114.654,Z 541.686,A -85,B 0,C 180,E1 -26219.366,E2 -26219.366} C_VEL
LIN {X 0,Y 119.047,Z 536.89,A -85,B 0,C 180,E1 -26224.259,E2 -26224.259} C_VEL
LIN {X 0,Y 124.964,Z 530.227,A -85,B 0,C 180,E1 -26229.25,E2 -26229.25} C_VEL
LIN {X 0,Y 131.907,Z 521.792,A -85,B 0,C 180,E1 -26233.84,E2 -26233.84} C_VEL
LIN {X 0,Y 138.443,Z 512.987,A -85,B 0,C 180,E1 -26237.4,E2 -26237.4} C_VEL
LIN {X 0,Y 141.572,Z 508.459,A -85,B 0,C 180,E1 -26238.873,E2 -26238.873} C_VEL
LIN {X 0,Y 142.173,Z 507.228,A -85,B 0,C 180,E1 -26239.345,E2 -26239.345} C_VEL
LIN {X 0,Y 143.955,Z 499.599,A -85,B 0,C 180,E1 -26242.945,E2 -26242.945} C_VEL
LIN {X 0,Y 144.52,Z 493.955,A -85,B 0,C 180,E1 -26245.763,E2 -26245.763} C_VEL
LIN {X 0,Y 144.115,Z 488.115,A -85,B 0,C 180,E1 -26249.199,E2 -26249.199} C_VEL
LIN {X 0,Y 143.319,Z 482.7,A -85,B 0,C 180,E1 -26252.762,E2 -26252.762} C_VEL
LIN {X 0,Y 142.667,Z 479.315,A -85,B 0,C 180,E1 -26255.235,E2 -26255.235} C_VEL
LIN {X 0,Y 141.728,Z 475.844,A -85,B 0,C 180,E1 -26258.166,E2 -26258.166} C_VEL
LIN {X 0,Y 140.212,Z 471.98,A -85,B 0,C 180,E1 -26262.497,E2 -26262.497} C_VEL
LIN {X 0,Y 139.286,Z 469.913,A -85,B 0,C 180,E1 -26265.387,E2 -26265.387} C_VEL
LIN {X 0,Y 137.844,Z 465.208,A -85,B 0,C 180,E1 -26274.147,E2 -26274.147} C_VEL
LIN {X 0,Y 137.526,Z 464.426,A -85,B 0,C 180,E1 -26280,E2 -26280} C_VEL
LIN {X 0,Y 137.636,Z 464.645,A -85,B 0,C 180,E1 -26282.927,E2 -26282.927} C_VEL
LIN {X 0,Y 137.919,Z 465.284,A -85,B 0,C 180,E1 -26285.849,E2 -26285.849} C_VEL
LIN {X 0,Y 139.503,Z 470.088,A -85,B 0,C 180,E1 -26294.589,E2 -26294.589} C_VEL
LIN {X 0,Y 140.802,Z 473.8,A -85,B 0,C 180,E1 -26298.93,E2 -26298.93} C_VEL
LIN {X 0,Y 141.693,Z 476.859,A -85,B 0,C 180,E1 -26301.839,E2 -26301.839} C_VEL
LIN {X 0,Y 142.902,Z 482.709,A -85,B 0,C 180,E1 -26306.271,E2 -26306.271} C_VEL
LIN {X 0,Y 143.937,Z 489.765,A -85,B 0,C 180,E1 -26310.842,E2 -26310.842} C_VEL
LIN {X 0,Y 144.194,Z 495.442,A -85,B 0,C 180,E1 -26314.046,E2 -26314.046} C_VEL
LIN {X 0,Y 143.514,Z 500.304,A -85,B 0,C 180,E1 -26316.337,E2 -26316.337} C_VEL
LIN {X 0,Y 141.79,Z 507.415,A -85,B 0,C 180,E1 -26319.535,E2 -26319.535} C_VEL
LIN {X 0,Y 140.346,Z 511.423,A -85,B 0,C 180,E1 -26321.31,E2 -26321.31} C_VEL
LIN {X 0,Y 133.547,Z 520.843,A -85,B 0,C 180,E1 -26324.728,E2 -26324.728} C_VEL
LIN {X 0,Y 126.41,Z 529.815,A -85,B 0,C 180,E1 -26329.211,E2 -26329.211} C_VEL
LIN {X 0,Y 120.089,Z 537.068,A -85,B 0,C 180,E1 -26334.18,E2 -26334.18} C_VEL
LIN {X 0,Y 115.937,Z 541.61,A -85,B 0,C 180,E1 -26338.293,E2 -26338.293} C_VEL
LIN {X 0,Y 111.768,Z 546.222,A -85,B 0,C 180,E1 -26343.885,E2 -26343.885} C_VEL
LIN {X 0,Y 107.91,Z 550.341,A -85,B 0,C 180,E1 -26350.995,E2 -26350.995} C_VEL
LIN {X 0,Y 105.774,Z 553.032,A -85,B 0,C 180,E1 -26358.502,E2 -26358.502} C_VEL
LIN {X 0,Y 104.963,Z 554.361,A -85,B 0,C 180,E1 -26366.16,E2 -26366.16} C_VEL
LIN {X 0,Y 105.033,Z 554.523,A -85,B 0,C 180,E1 -26370,E2 -26370} C_VEL
LIN {X 0,Y 105.222,Z 553.84,A -85,B 0,C 180,E1 -26377.676,E2 -26377.676} C_VEL
LIN {X 0,Y 106.669,Z 551.813,A -85,B 0,C 180,E1 -26385.28,E2 -26385.28} C_VEL
LIN {X 0,Y 109.643,Z 548.395,A -85,B 0,C 180,E1 -26392.618,E2 -26392.618} C_VEL
LIN {X 0,Y 114.229,Z 543.486,A -85,B 0,C 180,E1 -26399.485,E2 -26399.485} C_VEL
LIN {X 0,Y 120.083,Z 536.938,A -85,B 0,C 180,E1 -26405.821,E2 -26405.821} C_VEL
LIN {X 0,Y 126.406,Z 529.656,A -85,B 0,C 180,E1 -26410.789,E2 -26410.789} C_VEL
LIN {X 0,Y 133.553,Z 520.63,A -85,B 0,C 180,E1 -26415.268,E2 -26415.268} C_VEL
LIN {X 0,Y 140.303,Z 511.165,A -85,B 0,C 180,E1 -26418.709,E2 -26418.709} C_VEL
LIN {X 0,Y 142.155,Z 505.486,A -85,B 0,C 180,E1 -26421.238,E2 -26421.238} C_VEL
LIN {X 0,Y 143.809,Z 498.063,A -85,B 0,C 180,E1 -26424.564,E2 -26424.564} C_VEL
LIN {X 0,Y 144.101,Z 493.738,A -85,B 0,C 180,E1 -26426.724,E2 -26426.724} C_VEL
LIN {X 0,Y 143.502,Z 487.08,A -85,B 0,C 180,E1 -26430.676,E2 -26430.676} C_VEL
LIN {X 0,Y 142.531,Z 481.172,A -85,B 0,C 180,E1 -26434.641,E2 -26434.641} C_VEL
LIN {X 0,Y 141.529,Z 476.664,A -85,B 0,C 180,E1 -26438.134,E2 -26438.134} C_VEL
LIN {X 0,Y 140.162,Z 472.243,A -85,B 0,C 180,E1 -26442.491,E2 -26442.491} C_VEL
LIN {X 0,Y 139.302,Z 469.9,A -85,B 0,C 180,E1 -26445.389,E2 -26445.389} C_VEL
LIN {X 0,Y 137.683,Z 465.097,A -85,B 0,C 180,E1 -26454.141,E2 -26454.141} C_VEL
LIN {X 0,Y 137.264,Z 464.27,A -85,B 0,C 180,E1 -26460,E2 -26460} C_VEL
LIN {X 0,Y 137.587,Z 465.02,A -85,B 0,C 180,E1 -26465.864,E2 -26465.864} C_VEL
LIN {X 0,Y 139.054,Z 469.681,A -85,B 0,C 180,E1 -26474.638,E2 -26474.638} C_VEL
LIN {X 0,Y 139.501,Z 470.839,A -85,B 0,C 180,E1 -26476.226,E2 -26476.226} C_VEL
LIN {X 0,Y 139.926,Z 473.157,A -85,B 0,C 180,E1 -26478.448,E2 -26478.448} C_VEL
LIN {X 0,Y 139.825,Z 476.355,A -85,B 0,C 180,E1 -26480.505,E2 -26480.505} C_VEL
LIN {X 0,Y 138.62,Z 486.174,A -85,B 0,C 180,E1 -26485.781,E2 -26485.781} C_VEL
LIN {X 0,Y 138.648,Z 488.344,A -85,B 0,C 180,E1 -26487.197,E2 -26487.197} C_VEL
LIN {X 0,Y 139.083,Z 494.194,A -85,B 0,C 180,E1 -26491.193,E2 -26491.193} C_VEL
LIN {X 0,Y 138.838,Z 499.521,A -85,B 0,C 180,E1 -26494.354,E2 -26494.354} C_VEL
LIN {X 0,Y 137.594,Z 505.23,A -85,B 0,C 180,E1 -26497.266,E2 -26497.266} C_VEL
LIN {X 0,Y 136.198,Z 509.359,A -85,B 0,C 180,E1 -26499.284,E2 -26499.284} C_VEL
LIN {X 0,Y 129.117,Z 518.809,A -85,B 0,C 180,E1 -26502.708,E2 -26502.708} C_VEL
LIN {X 0,Y 121.6,Z 527.815,A -85,B 0,C 180,E1 -26507.227,E2 -26507.227} C_VEL
LIN {X 0,Y 114.843,Z 535.074,A -85,B 0,C 180,E1 -26512.269,E2 -26512.269} C_VEL
LIN {X 0,Y 109.991,Z 540.154,A -85,B 0,C 180,E1 -26517.104,E2 -26517.104} C_VEL
LIN {X 0,Y 105.829,Z 544.226,A -85,B 0,C 180,E1 -26522.299,E2 -26522.299} C_VEL
LIN {X 0,Y 101.572,Z 548.349,A -85,B 0,C 180,E1 -26529.76,E2 -26529.76} C_VEL
LIN {X 0,Y 99.056,Z 551.039,A -85,B 0,C 180,E1 -26537.711,E2 -26537.711} C_VEL
LIN {X 0,Y 97.961,Z 552.38,A -85,B 0,C 180,E1 -26545.886,E2 -26545.886} C_VEL
LIN {X 0,Y 98.006,Z 552.553,A -85,B 0,C 180,E1 -26550,E2 -26550} C_VEL
LIN {X 0,Y 98.331,Z 551.917,A -85,B 0,C 180,E1 -26558.219,E2 -26558.219} C_VEL
LIN {X 0,Y 100.08,Z 549.946,A -85,B 0,C 180,E1 -26566.314,E2 -26566.314} C_VEL
LIN {X 0,Y 103.413,Z 546.593,A -85,B 0,C 180,E1 -26574.065,E2 -26574.065} C_VEL
LIN {X 0,Y 108.482,Z 541.754,A -85,B 0,C 180,E1 -26581.218,E2 -26581.218} C_VEL
LIN {X 0,Y 113.817,Z 536.337,A -85,B 0,C 180,E1 -26586.828,E2 -26586.828} C_VEL
LIN {X 0,Y 120.543,Z 529.181,A -85,B 0,C 180,E1 -26592.105,E2 -26592.105} C_VEL
LIN {X 0,Y 127.97,Z 520.507,A -85,B 0,C 180,E1 -26596.693,E2 -26596.693} C_VEL
LIN {X 0,Y 134.951,Z 511.428,A -85,B 0,C 180,E1 -26600.189,E2 -26600.189} C_VEL
LIN {X 0,Y 136.146,Z 509.76,A -85,B 0,C 180,E1 -26600.744,E2 -26600.744} C_VEL
LIN {X 0,Y 137.23,Z 506.903,A -85,B 0,C 180,E1 -26602.08,E2 -26602.08} C_VEL
LIN {X 0,Y 138.599,Z 501.578,A -85,B 0,C 180,E1 -26604.772,E2 -26604.772} C_VEL
LIN {X 0,Y 139.156,Z 497.296,A -85,B 0,C 180,E1 -26607.118,E2 -26607.118} C_VEL
LIN {X 0,Y 139.027,Z 491.644,A -85,B 0,C 180,E1 -26610.748,E2 -26610.748} C_VEL
LIN {X 0,Y 138.489,Z 486.547,A -85,B 0,C 180,E1 -26614.446,E2 -26614.446} C_VEL
LIN {X 0,Y 137.901,Z 483.046,A -85,B 0,C 180,E1 -26617.37,E2 -26617.37} C_VEL
LIN {X 0,Y 137.544,Z 481.198,A -85,B 0,C 180,E1 -26619.042,E2 -26619.042} C_VEL
LIN {X 0,Y 136.299,Z 477.515,A -85,B 0,C 180,E1 -26623.525,E2 -26623.525} C_VEL
LIN {X 0,Y 134.794,Z 473.296,A -85,B 0,C 180,E1 -26631.001,E2 -26631.001} C_VEL
LIN {X 0,Y 134.683,Z 471.775,A -85,B 0,C 180,E1 -26634.009,E2 -26634.009} C_VEL
LIN {X 0,Y 134.519,Z 471.059,A -85,B 0,C 180,E1 -26637.005,E2 -26637.005} C_VEL
LIN {X 0,Y 134.476,Z 470.839,A -85,B 0,C 180,E1 -26640,E2 -26640} C_VEL
LIN {X 0,Y 134.574,Z 471.074,A -85,B 0,C 180,E1 -26642.993,E2 -26642.993} C_VEL
LIN {X 0,Y 134.764,Z 471.861,A -85,B 0,C 180,E1 -26645.987,E2 -26645.987} C_VEL
LIN {X 0,Y 135.403,Z 474.967,A -85,B 0,C 180,E1 -26651.983,E2 -26651.983} C_VEL
LIN {X 0,Y 136.451,Z 477.924,A -85,B 0,C 180,E1 -26656.456,E2 -26656.456} C_VEL
LIN {X 0,Y 137.485,Z 482.19,A -85,B 0,C 180,E1 -26660.967,E2 -26660.967} C_VEL
LIN {X 0,Y 138.327,Z 487.901,A -85,B 0,C 180,E1 -26665.586,E2 -26665.586} C_VEL
LIN {X 0,Y 138.841,Z 493.898,A -85,B 0,C 180,E1 -26669.742,E2 -26669.742} C_VEL
LIN {X 0,Y 138.784,Z 499.228,A -85,B 0,C 180,E1 -26672.981,E2 -26672.981} C_VEL
LIN {X 0,Y 137.804,Z 503.909,A -85,B 0,C 180,E1 -26675.313,E2 -26675.313} C_VEL
LIN {X 0,Y 135.443,Z 511.353,A -85,B 0,C 180,E1 -26678.891,E2 -26678.891} C_VEL
LIN {X 0,Y 134.547,Z 513.036,A -85,B 0,C 180,E1 -26679.604,E2 -26679.604} C_VEL
LIN {X 0,Y 127.5,Z 522.151,A -85,B 0,C 180,E1 -26683.083,E2 -26683.083} C_VEL
LIN {X 0,Y 120.076,Z 530.865,A -85,B 0,C 180,E1 -26687.693,E2 -26687.693} C_VEL
LIN {X 0,Y 114.376,Z 537,A -85,B 0,C 180,E1 -26692.087,E2 -26692.087} C_VEL
LIN {X 0,Y 109.512,Z 541.962,A -85,B 0,C 180,E1 -26696.767,E2 -26696.767} C_VEL
LIN {X 0,Y 105.379,Z 546.154,A -85,B 0,C 180,E1 -26702.17,E2 -26702.17} C_VEL
LIN {X 0,Y 101.181,Z 550.272,A -85,B 0,C 180,E1 -26709.677,E2 -26709.677} C_VEL
LIN {X 0,Y 98.791,Z 552.963,A -85,B 0,C 180,E1 -26717.677,E2 -26717.677} C_VEL
LIN {X 0,Y 97.891,Z 554.292,A -85,B 0,C 180,E1 -26725.883,E2 -26725.883} C_VEL
LIN {X 0,Y 97.94,Z 554.455,A -85,B 0,C 180,E1 -26730,E2 -26730} C_VEL
LIN {X 0,Y 98.179,Z 553.77,A -85,B 0,C 180,E1 -26738.231,E2 -26738.231} C_VEL
LIN {X 0,Y 99.791,Z 551.743,A -85,B 0,C 180,E1 -26746.362,E2 -26746.362} C_VEL
LIN {X 0,Y 103.107,Z 548.325,A -85,B 0,C 180,E1 -26754.14,E2 -26754.14} C_VEL
LIN {X 0,Y 108.072,Z 543.415,A -85,B 0,C 180,E1 -26761.348,E2 -26761.348} C_VEL
LIN {X 0,Y 114.367,Z 536.867,A -85,B 0,C 180,E1 -26767.916,E2 -26767.916} C_VEL
LIN {X 0,Y 121.09,Z 529.585,A -85,B 0,C 180,E1 -26772.997,E2 -26772.997} C_VEL
LIN {X 0,Y 128.644,Z 520.559,A -85,B 0,C 180,E1 -26777.52,E2 -26777.52} C_VEL
LIN {X 0,Y 134.525,Z 512.795,A -85,B 0,C 180,E1 -26780.406,E2 -26780.406} C_VEL
LIN {X 0,Y 135.996,Z 509.298,A -85,B 0,C 180,E1 -26782.005,E2 -26782.005} C_VEL
LIN {X 0,Y 138.09,Z 502.291,A -85,B 0,C 180,E1 -26785.372,E2 -26785.372} C_VEL
LIN {X 0,Y 138.798,Z 497.494,A -85,B 0,C 180,E1 -26787.884,E2 -26787.884} C_VEL
LIN {X 0,Y 138.661,Z 492.441,A -85,B 0,C 180,E1 -26791.066,E2 -26791.066} C_VEL
LIN {X 0,Y 137.942,Z 485.686,A -85,B 0,C 180,E1 -26795.947,E2 -26795.947} C_VEL
LIN {X 0,Y 137.335,Z 481.983,A -85,B 0,C 180,E1 -26799.009,E2 -26799.009} C_VEL
LIN {X 0,Y 136.666,Z 478.984,A -85,B 0,C 180,E1 -26802.028,E2 -26802.028} C_VEL
LIN {X 0,Y 135.892,Z 476.62,A -85,B 0,C 180,E1 -26805.014,E2 -26805.014} C_VEL
LIN {X 0,Y 134.626,Z 472.257,A -85,B 0,C 180,E1 -26812.689,E2 -26812.689} C_VEL
LIN {X 0,Y 134.551,Z 471.656,A -85,B 0,C 180,E1 -26814.004,E2 -26814.004} C_VEL
LIN {X 0,Y 134.232,Z 470.669,A -85,B 0,C 180,E1 -26820,E2 -26820} C_VEL
LIN {X 0,Y 134.254,Z 470.92,A -85,B 0,C 180,E1 -26823.001,E2 -26823.001} C_VEL
LIN {X 0,Y 134.466,Z 471.912,A -85,B 0,C 180,E1 -26826.76,E2 -26826.76} C_VEL
LIN {X 0,Y 135.667,Z 476.308,A -85,B 0,C 180,E1 -26835.012,E2 -26835.012} C_VEL
LIN {X 0,Y 136.916,Z 479.626,A -85,B 0,C 180,E1 -26839.491,E2 -26839.491} C_VEL
LIN {X 0,Y 137.747,Z 482.719,A -85,B 0,C 180,E1 -26842.657,E2 -26842.657} C_VEL
LIN {X 0,Y 138.648,Z 488.344,A -85,B 0,C 180,E1 -26847.197,E2 -26847.197} C_VEL
LIN {X 0,Y 138.654,Z 490.522,A -85,B 0,C 180,E1 -26848.571,E2 -26848.571} C_VEL
LIN {X 0,Y 137.924,Z 494.336,A -85,B 0,C 180,E1 -26850.462,E2 -26850.462} C_VEL
LIN {X 0,Y 136.55,Z 498.443,A -85,B 0,C 180,E1 -26852.196,E2 -26852.196} C_VEL
LIN {X 0,Y 134.041,Z 504.16,A -85,B 0,C 180,E1 -26854.441,E2 -26854.441} C_VEL
LIN {X 0,Y 131.28,Z 509.686,A -85,B 0,C 180,E1 -26856.77,E2 -26856.77} C_VEL
LIN {X 0,Y 130.553,Z 511.133,A -85,B 0,C 180,E1 -26857.437,E2 -26857.437} C_VEL
LIN {X 0,Y 123.226,Z 520.272,A -85,B 0,C 180,E1 -26860.914,E2 -26860.914} C_VEL
LIN {X 0,Y 115.393,Z 529,A -85,B 0,C 180,E1 -26865.541,E2 -26865.541} C_VEL
LIN {X 0,Y 108.107,Z 536.292,A -85,B 0,C 180,E1 -26870.993,E2 -26870.993} C_VEL
LIN {X 0,Y 102.473,Z 541.661,A -85,B 0,C 180,E1 -26876.725,E2 -26876.725} C_VEL
LIN {X 0,Y 96.973,Z 546.544,A -85,B 0,C 180,E1 -26884.225,E2 -26884.225} C_VEL
LIN {X 0,Y 93.309,Z 549.936,A -85,B 0,C 180,E1 -26892.466,E2 -26892.466} C_VEL
LIN {X 0,Y 91.319,Z 551.944,A -85,B 0,C 180,E1 -26901.146,E2 -26901.146} C_VEL
LIN {X 0,Y 90.914,Z 552.622,A -85,B 0,C 180,E1 -26910,E2 -26910} C_VEL
LIN {X 0,Y 91.312,Z 551.986,A -85,B 0,C 180,E1 -26918.855,E2 -26918.855} C_VEL
LIN {X 0,Y 93.278,Z 550.014,A -85,B 0,C 180,E1 -26927.541,E2 -26927.541} C_VEL
LIN {X 0,Y 96.953,Z 546.661,A -85,B 0,C 180,E1 -26935.781,E2 -26935.781} C_VEL
LIN {X 0,Y 102.443,Z 541.823,A -85,B 0,C 180,E1 -26943.288,E2 -26943.288} C_VEL
LIN {X 0,Y 107.41,Z 537.178,A -85,B 0,C 180,E1 -26948.4,E2 -26948.4} C_VEL
LIN {X 0,Y 114.292,Z 530.361,A -85,B 0,C 180,E1 -26953.772,E2 -26953.772} C_VEL
LIN {X 0,Y 122.036,Z 521.926,A -85,B 0,C 180,E1 -26958.475,E2 -26958.475} C_VEL
LIN {X 0,Y 129.256,Z 513.119,A -85,B 0,C 180,E1 -26962.037,E2 -26962.037} C_VEL
LIN {X 0,Y 130.514,Z 511.494,A -85,B 0,C 180,E1 -26962.587,E2 -26962.587} C_VEL
LIN {X 0,Y 131.421,Z 509.831,A -85,B 0,C 180,E1 -26963.337,E2 -26963.337} C_VEL
LIN {X 0,Y 133.154,Z 504.31,A -85,B 0,C 180,E1 -26966.322,E2 -26966.322} C_VEL
LIN {X 0,Y 133.909,Z 499.817,A -85,B 0,C 180,E1 -26969.048,E2 -26969.048} C_VEL
LIN {X 0,Y 133.954,Z 494.145,A -85,B 0,C 180,E1 -26973.116,E2 -26973.116} C_VEL
LIN {X 0,Y 133.596,Z 489.008,A -85,B 0,C 180,E1 -26977.381,E2 -26977.381} C_VEL
LIN {X 0,Y 133.195,Z 486.421,A -85,B 0,C 180,E1 -26979.942,E2 -26979.942} C_VEL
LIN {X 0,Y 132.211,Z 482.931,A -85,B 0,C 180,E1 -26984.586,E2 -26984.586} C_VEL
LIN {X 0,Y 131.211,Z 478.18,A -85,B 0,C 180,E1 -26993.85,E2 -26993.85} C_VEL
LIN {X 0,Y 131.142,Z 477.349,A -85,B 0,C 180,E1 -26996.928,E2 -26996.928} C_VEL
LIN {X 0,Y 131.125,Z 477.103,A -85,B 0,C 180,E1 -27000,E2 -27000} C_VEL
LIN {X 0,Y 131.208,Z 477.355,A -85,B 0,C 180,E1 -27003.07,E2 -27003.07} C_VEL
LIN {X 0,Y 131.291,Z 478.289,A -85,B 0,C 180,E1 -27006.146,E2 -27006.146} C_VEL
LIN {X 0,Y 131.806,Z 481.364,A -85,B 0,C 180,E1 -27012.315,E2 -27012.315} C_VEL
LIN {X 0,Y 132.386,Z 483.272,A -85,B 0,C 180,E1 -27015.393,E2 -27015.393} C_VEL
LIN {X 0,Y 133.121,Z 487.369,A -85,B 0,C 180,E1 -27020.069,E2 -27020.069} C_VEL
LIN {X 0,Y 133.578,Z 492.956,A -85,B 0,C 180,E1 -27024.892,E2 -27024.892} C_VEL
LIN {X 0,Y 133.697,Z 497.447,A -85,B 0,C 180,E1 -27028.235,E2 -27028.235} C_VEL
LIN {X 0,Y 133.345,Z 502.854,A -85,B 0,C 180,E1 -27031.807,E2 -27031.807} C_VEL
LIN {X 0,Y 131.954,Z 507.692,A -85,B 0,C 180,E1 -27034.355,E2 -27034.355} C_VEL
LIN {X 0,Y 129.949,Z 512.911,A -85,B 0,C 180,E1 -27037.043,E2 -27037.043} C_VEL
LIN {X 0,Y 127.551,Z 516.314,A -85,B 0,C 180,E1 -27038.333,E2 -27038.333} C_VEL
LIN {X 0,Y 120.414,Z 524.795,A -85,B 0,C 180,E1 -27041.912,E2 -27041.912} C_VEL
LIN {X 0,Y 112.815,Z 532.995,A -85,B 0,C 180,E1 -27046.743,E2 -27046.743} C_VEL
LIN {X 0,Y 106.966,Z 538.745,A -85,B 0,C 180,E1 -27051.378,E2 -27051.378} C_VEL
LIN {X 0,Y 100.485,Z 544.841,A -85,B 0,C 180,E1 -27058.361,E2 -27058.361} C_VEL
LIN {X 0,Y 96.627,Z 548.33,A -85,B 0,C 180,E1 -27064.125,E2 -27064.125} C_VEL
LIN {X 0,Y 92.966,Z 551.722,A -85,B 0,C 180,E1 -27072.398,E2 -27072.398} C_VEL
LIN {X 0,Y 91.139,Z 553.727,A -85,B 0,C 180,E1 -27081.128,E2 -27081.128} C_VEL
LIN {X 0,Y 90.84,Z 554.386,A -85,B 0,C 180,E1 -27090,E2 -27090} C_VEL
LIN {X 0,Y 91.139,Z 553.701,A -85,B 0,C 180,E1 -27098.872,E2 -27098.872} C_VEL
LIN {X 0,Y 92.964,Z 551.673,A -85,B 0,C 180,E1 -27107.601,E2 -27107.601} C_VEL
LIN {X 0,Y 96.628,Z 548.255,A -85,B 0,C 180,E1 -27115.874,E2 -27115.874} C_VEL
LIN {X 0,Y 102.037,Z 543.345,A -85,B 0,C 180,E1 -27123.436,E2 -27123.436} C_VEL
LIN {X 0,Y 108.821,Z 536.796,A -85,B 0,C 180,E1 -27130.228,E2 -27130.228} C_VEL
LIN {X 0,Y 115.972,Z 529.514,A -85,B 0,C 180,E1 -27135.402,E2 -27135.402} C_VEL
LIN {X 0,Y 123.954,Z 520.488,A -85,B 0,C 180,E1 -27139.945,E2 -27139.945} C_VEL
LIN {X 0,Y 128.663,Z 514.625,A -85,B 0,C 180,E1 -27142.162,E2 -27142.162} C_VEL
LIN {X 0,Y 129.808,Z 512.828,A -85,B 0,C 180,E1 -27142.91,E2 -27142.91} C_VEL
LIN {X 0,Y 132.25,Z 506.286,A -85,B 0,C 180,E1 -27146.268,E2 -27146.268} C_VEL
LIN {X 0,Y 133.184,Z 502.76,A -85,B 0,C 180,E1 -27148.151,E2 -27148.151} C_VEL
LIN {X 0,Y 133.563,Z 498.955,A -85,B 0,C 180,E1 -27150.537,E2 -27150.537} C_VEL
LIN {X 0,Y 133.426,Z 492.8,A -85,B 0,C 180,E1 -27155.078,E2 -27155.078} C_VEL
LIN {X 0,Y 133.108,Z 488.966,A -85,B 0,C 180,E1 -27158.31,E2 -27158.31} C_VEL
LIN {X 0,Y 132.977,Z 487.166,A -85,B 0,C 180,E1 -27159.908,E2 -27159.908} C_VEL
LIN {X 0,Y 132.568,Z 484.672,A -85,B 0,C 180,E1 -27162.603,E2 -27162.603} C_VEL
LIN {X 0,Y 132.186,Z 483.123,A -85,B 0,C 180,E1 -27164.584,E2 -27164.584} C_VEL
LIN {X 0,Y 131.264,Z 479.521,A -85,B 0,C 180,E1 -27170.757,E2 -27170.757} C_VEL
LIN {X 0,Y 131.119,Z 478.032,A -85,B 0,C 180,E1 -27173.846,E2 -27173.846} C_VEL
LIN {X 0,Y 130.929,Z 477.28,A -85,B 0,C 180,E1 -27176.923,E2 -27176.923} C_VEL
LIN {X 0,Y 130.888,Z 476.941,A -85,B 0,C 180,E1 -27180,E2 -27180} C_VEL
LIN {X 0,Y 130.888,Z 477.209,A -85,B 0,C 180,E1 -27183.078,E2 -27183.078} C_VEL
LIN {X 0,Y 131.012,Z 477.934,A -85,B 0,C 180,E1 -27186.159,E2 -27186.159} C_VEL
LIN {X 0,Y 131.402,Z 480.96,A -85,B 0,C 180,E1 -27192.354,E2 -27192.354} C_VEL
LIN {X 0,Y 132.369,Z 483.86,A -85,B 0,C 180,E1 -27197.12,E2 -27197.12} C_VEL
LIN {X 0,Y 133.006,Z 486.182,A -85,B 0,C 180,E1 -27200.088,E2 -27200.088} C_VEL
LIN {X 0,Y 133.537,Z 489.552,A -85,B 0,C 180,E1 -27203.383,E2 -27203.383} C_VEL
LIN {X 0,Y 133.81,Z 493.647,A -85,B 0,C 180,E1 -27206.764,E2 -27206.764} C_VEL
LIN {X 0,Y 133.786,Z 499.379,A -85,B 0,C 180,E1 -27210.883,E2 -27210.883} C_VEL
LIN {X 0,Y 133.515,Z 502.077,A -85,B 0,C 180,E1 -27212.626,E2 -27212.626} C_VEL
LIN {X 0,Y 132.259,Z 506.925,A -85,B 0,C 180,E1 -27215.317,E2 -27215.317} C_VEL
LIN {X 0,Y 131.28,Z 509.686,A -85,B 0,C 180,E1 -27216.77,E2 -27216.77} C_VEL
LIN {X 0,Y 129.595,Z 512.318,A -85,B 0,C 180,E1 -27217.799,E2 -27217.799} C_VEL
LIN {X 0,Y 127.314,Z 514.972,A -85,B 0,C 180,E1 -27218.595,E2 -27218.595} C_VEL
LIN {X 0,Y 121.726,Z 519.977,A -85,B 0,C 180,E1 -27219.785,E2 -27219.785} C_VEL
LIN {X 0,Y 114.151,Z 525.888,A -85,B 0,C 180,E1 -27221.4,E2 -27221.4} C_VEL
LIN {X 0,Y 110.287,Z 529.204,A -85,B 0,C 180,E1 -27223.037,E2 -27223.037} C_VEL
LIN {X 0,Y 103.958,Z 535.215,A -85,B 0,C 180,E1 -27227.465,E2 -27227.465} C_VEL
LIN {X 0,Y 98.318,Z 540.295,A -85,B 0,C 180,E1 -27232.584,E2 -27232.584} C_VEL
LIN {X 0,Y 93.456,Z 544.366,A -85,B 0,C 180,E1 -27238.237,E2 -27238.237} C_VEL
LIN {X 0,Y 88.305,Z 548.489,A -85,B 0,C 180,E1 -27246.551,E2 -27246.551} C_VEL
LIN {X 0,Y 85.209,Z 551.178,A -85,B 0,C 180,E1 -27255.674,E2 -27255.674} C_VEL
LIN {X 0,Y 83.812,Z 552.518,A -85,B 0,C 180,E1 -27265.19,E2 -27265.19} C_VEL
LIN {X 0,Y 83.813,Z 552.691,A -85,B 0,C 180,E1 -27270,E2 -27270} C_VEL
LIN {X 0,Y 84.295,Z 552.055,A -85,B 0,C 180,E1 -27279.599,E2 -27279.599} C_VEL
LIN {X 0,Y 86.495,Z 550.083,A -85,B 0,C 180,E1 -27288.967,E2 -27288.967} C_VEL
LIN {X 0,Y 90.599,Z 546.729,A -85,B 0,C 180,E1 -27297.739,E2 -27297.739} C_VEL
LIN {X 0,Y 96.56,Z 541.891,A -85,B 0,C 180,E1 -27305.611,E2 -27305.611} C_VEL
LIN {X 0,Y 101.758,Z 537.4,A -85,B 0,C 180,E1 -27310.744,E2 -27310.744} C_VEL
LIN {X 0,Y 109.264,Z 530.429,A -85,B 0,C 180,E1 -27316.354,E2 -27316.354} C_VEL
LIN {X 0,Y 117.425,Z 521.993,A -85,B 0,C 180,E1 -27321.085,E2 -27321.085} C_VEL
LIN {X 0,Y 124.965,Z 513.24,A -85,B 0,C 180,E1 -27324.589,E2 -27324.589} C_VEL
LIN {X 0,Y 126.178,Z 511.315,A -85,B 0,C 180,E1 -27325.459,E2 -27325.459} C_VEL
LIN {X 0,Y 128.039,Z 506.056,A -85,B 0,C 180,E1 -27328.57,E2 -27328.57} C_VEL
LIN {X 0,Y 128.611,Z 502.592,A -85,B 0,C 180,E1 -27330.966,E2 -27330.966} C_VEL
LIN {X 0,Y 128.899,Z 498.534,A -85,B 0,C 180,E1 -27334.139,E2 -27334.139} C_VEL
LIN {X 0,Y 128.91,Z 494.257,A -85,B 0,C 180,E1 -27337.945,E2 -27337.945} C_VEL
LIN {X 0,Y 128.678,Z 491.514,A -85,B 0,C 180,E1 -27340.87,E2 -27340.87} C_VEL
LIN {X 0,Y 128.2,Z 489.2,A -85,B 0,C 180,E1 -27344.091,E2 -27344.091} C_VEL
LIN {X 0,Y 127.396,Z 485.875,A -85,B 0,C 180,E1 -27350.473,E2 -27350.473} C_VEL
LIN {X 0,Y 127.426,Z 484.429,A -85,B 0,C 180,E1 -27353.667,E2 -27353.667} C_VEL
LIN {X 0,Y 127.459,Z 483.494,A -85,B 0,C 180,E1 -27356.839,E2 -27356.839} C_VEL
LIN {X 0,Y 127.494,Z 483.185,A -85,B 0,C 180,E1 -27360,E2 -27360} C_VEL
LIN {X 0,Y 127.533,Z 483.501,A -85,B 0,C 180,E1 -27363.159,E2 -27363.159} C_VEL
LIN {X 0,Y 127.503,Z 484.926,A -85,B 0,C 180,E1 -27367.175,E2 -27367.175} C_VEL
LIN {X 0,Y 128.112,Z 488.549,A -85,B 0,C 180,E1 -27374.292,E2 -27374.292} C_VEL
LIN {X 0,Y 128.59,Z 492.413,A -85,B 0,C 180,E1 -27379.143,E2 -27379.143} C_VEL
LIN {X 0,Y 128.644,Z 497.884,A -85,B 0,C 180,E1 -27384.188,E2 -27384.188} C_VEL
LIN {X 0,Y 128.423,Z 502.461,A -85,B 0,C 180,E1 -27387.812,E2 -27387.812} C_VEL
LIN {X 0,Y 127.92,Z 506.115,A -85,B 0,C 180,E1 -27390.396,E2 -27390.396} C_VEL
LIN {X 0,Y 126.039,Z 511.204,A -85,B 0,C 180,E1 -27393.236,E2 -27393.236} C_VEL
LIN {X 0,Y 124.746,Z 514.106,A -85,B 0,C 180,E1 -27394.859,E2 -27394.859} C_VEL
LIN {X 0,Y 123.024,Z 516.539,A -85,B 0,C 180,E1 -27395.844,E2 -27395.844} C_VEL
LIN {X 0,Y 114.59,Z 525.986,A -85,B 0,C 180,E1 -27399.945,E2 -27399.945} C_VEL
LIN {X 0,Y 106.638,Z 533.937,A -85,B 0,C 180,E1 -27404.888,E2 -27404.888} C_VEL
LIN {X 0,Y 99.561,Z 540.339,A -85,B 0,C 180,E1 -27410.557,E2 -27410.557} C_VEL
LIN {X 0,Y 92.953,Z 546.017,A -85,B 0,C 180,E1 -27418.044,E2 -27418.044} C_VEL
LIN {X 0,Y 87.924,Z 550.135,A -85,B 0,C 180,E1 -27426.442,E2 -27426.442} C_VEL
LIN {X 0,Y 84.931,Z 552.826,A -85,B 0,C 180,E1 -27435.626,E2 -27435.626} C_VEL
LIN {X 0,Y 83.739,Z 554.155,A -85,B 0,C 180,E1 -27445.185,E2 -27445.185} C_VEL
LIN {X 0,Y 83.761,Z 554.317,A -85,B 0,C 180,E1 -27450,E2 -27450} C_VEL
LIN {X 0,Y 84.125,Z 553.632,A -85,B 0,C 180,E1 -27459.618,E2 -27459.618} C_VEL
LIN {X 0,Y 86.196,Z 551.603,A -85,B 0,C 180,E1 -27469.034,E2 -27469.034} C_VEL
LIN {X 0,Y 90.258,Z 548.185,A -85,B 0,C 180,E1 -27477.852,E2 -27477.852} C_VEL
LIN {X 0,Y 96.134,Z 543.274,A -85,B 0,C 180,E1 -27485.792,E2 -27485.792} C_VEL
LIN {X 0,Y 103.469,Z 536.726,A -85,B 0,C 180,E1 -27492.783,E2 -27492.783} C_VEL
LIN {X 0,Y 111.086,Z 529.443,A -85,B 0,C 180,E1 -27498.02,E2 -27498.02} C_VEL
LIN {X 0,Y 119.506,Z 520.416,A -85,B 0,C 180,E1 -27502.553,E2 -27502.553} C_VEL
LIN {X 0,Y 123.907,Z 515.149,A -85,B 0,C 180,E1 -27504.575,E2 -27504.575} C_VEL
LIN {X 0,Y 125.265,Z 512.612,A -85,B 0,C 180,E1 -27505.872,E2 -27505.872} C_VEL
LIN {X 0,Y 127.355,Z 507.376,A -85,B 0,C 180,E1 -27508.764,E2 -27508.764} C_VEL
LIN {X 0,Y 128.208,Z 503.431,A -85,B 0,C 180,E1 -27511.291,E2 -27511.291} C_VEL
LIN {X 0,Y 128.475,Z 498.758,A -85,B 0,C 180,E1 -27514.916,E2 -27514.916} C_VEL
LIN {X 0,Y 128.486,Z 494.746,A -85,B 0,C 180,E1 -27518.415,E2 -27518.415} C_VEL
LIN {X 0,Y 128.329,Z 491.224,A -85,B 0,C 180,E1 -27522.009,E2 -27522.009} C_VEL
LIN {X 0,Y 127.923,Z 488.391,A -85,B 0,C 180,E1 -27525.687,E2 -27525.687} C_VEL
LIN {X 0,Y 127.362,Z 484.415,A -85,B 0,C 180,E1 -27533.342,E2 -27533.342} C_VEL
LIN {X 0,Y 127.274,Z 483.401,A -85,B 0,C 180,E1 -27536.835,E2 -27536.835} C_VEL
LIN {X 0,Y 127.257,Z 483.04,A -85,B 0,C 180,E1 -27540,E2 -27540} C_VEL
LIN {X 0,Y 127.226,Z 483.333,A -85,B 0,C 180,E1 -27543.167,E2 -27543.167} C_VEL
LIN {X 0,Y 127.249,Z 484.172,A -85,B 0,C 180,E1 -27546.342,E2 -27546.342} C_VEL
LIN {X 0,Y 127.494,Z 487.183,A -85,B 0,C 180,E1 -27552.738,E2 -27552.738} C_VEL
LIN {X 0,Y 128.292,Z 490.178,A -85,B 0,C 180,E1 -27557.682,E2 -27557.682} C_VEL
LIN {X 0,Y 128.732,Z 493.773,A -85,B 0,C 180,E1 -27561.86,E2 -27561.86} C_VEL
LIN {X 0,Y 128.769,Z 498.255,A -85,B 0,C 180,E1 -27565.889,E2 -27565.889} C_VEL
LIN {X 0,Y 128.46,Z 502.875,A -85,B 0,C 180,E1 -27569.498,E2 -27569.498} C_VEL
LIN {X 0,Y 127.701,Z 506.705,A -85,B 0,C 180,E1 -27572.063,E2 -27572.063} C_VEL
LIN {X 0,Y 126.011,Z 511.236,A -85,B 0,C 180,E1 -27574.671,E2 -27574.671} C_VEL
LIN {X 0,Y 124.973,Z 512.905,A -85,B 0,C 180,E1 -27575.436,E2 -27575.436} C_VEL
LIN {X 0,Y 117.473,Z 521.695,A -85,B 0,C 180,E1 -27578.946,E2 -27578.946} C_VEL
LIN {X 0,Y 110.287,Z 529.204,A -85,B 0,C 180,E1 -27583.037,E2 -27583.037} C_VEL
LIN {X 0,Y 106.643,Z 532.308,A -85,B 0,C 180,E1 -27584.881,E2 -27584.881} C_VEL
LIN {X 0,Y 99.478,Z 537.01,A -85,B 0,C 180,E1 -27587.657,E2 -27587.657} C_VEL
LIN {X 0,Y 92.433,Z 541.106,A -85,B 0,C 180,E1 -27591.017,E2 -27591.017} C_VEL
LIN {X 0,Y 89.114,Z 543.222,A -85,B 0,C 180,E1 -27593.792,E2 -27593.792} C_VEL
LIN {X 0,Y 84.388,Z 546.684,A -85,B 0,C 180,E1 -27600.021,E2 -27600.021} C_VEL
LIN {X 0,Y 79.816,Z 550.076,A -85,B 0,C 180,E1 -27609.378,E2 -27609.378} C_VEL
LIN {X 0,Y 77.298,Z 552.083,A -85,B 0,C 180,E1 -27619.523,E2 -27619.523} C_VEL
LIN {X 0,Y 76.735,Z 552.76,A -85,B 0,C 180,E1 -27630.001,E2 -27630.001} C_VEL
LIN {X 0,Y 77.29,Z 552.123,A -85,B 0,C 180,E1 -27640.479,E2 -27640.479} C_VEL
LIN {X 0,Y 79.777,Z 550.152,A -85,B 0,C 180,E1 -27650.634,E2 -27650.634} C_VEL
LIN {X 0,Y 84.371,Z 546.797,A -85,B 0,C 180,E1 -27659.987,E2 -27659.987} C_VEL
LIN {X 0,Y 90.858,Z 541.959,A -85,B 0,C 180,E1 -27668.23,E2 -27668.23} C_VEL
LIN {X 0,Y 96.458,Z 537.468,A -85,B 0,C 180,E1 -27673.515,E2 -27673.515} C_VEL
LIN {X 0,Y 104.467,Z 530.496,A -85,B 0,C 180,E1 -27679.187,E2 -27679.187} C_VEL
LIN {X 0,Y 113.081,Z 522.06,A -85,B 0,C 180,E1 -27683.897,E2 -27683.897} C_VEL
LIN {X 0,Y 120.407,Z 513.939,A -85,B 0,C 180,E1 -27687.16,E2 -27687.16} C_VEL
LIN {X 0,Y 121.786,Z 511.267,A -85,B 0,C 180,E1 -27688.709,E2 -27688.709} C_VEL
LIN {X 0,Y 122.918,Z 508,A -85,B 0,C 180,E1 -27690.897,E2 -27690.897} C_VEL
LIN {X 0,Y 123.762,Z 502.691,A -85,B 0,C 180,E1 -27695.311,E2 -27695.311} C_VEL
LIN {X 0,Y 123.986,Z 499.785,A -85,B 0,C 180,E1 -27698.099,E2 -27698.099} C_VEL
LIN {X 0,Y 124.013,Z 496.451,A -85,B 0,C 180,E1 -27701.838,E2 -27701.838} C_VEL
LIN {X 0,Y 123.685,Z 494.407,A -85,B 0,C 180,E1 -27705.012,E2 -27705.012} C_VEL
LIN {X 0,Y 123.365,Z 490.445,A -85,B 0,C 180,E1 -27713.457,E2 -27713.457} C_VEL
LIN {X 0,Y 123.488,Z 489.46,A -85,B 0,C 180,E1 -27716.737,E2 -27716.737} C_VEL
LIN {X 0,Y 123.568,Z 489.111,A -85,B 0,C 180,E1 -27720,E2 -27720} C_VEL
LIN {X 0,Y 123.557,Z 489.487,A -85,B 0,C 180,E1 -27723.261,E2 -27723.261} C_VEL
LIN {X 0,Y 123.456,Z 490.574,A -85,B 0,C 180,E1 -27726.537,E2 -27726.537} C_VEL
LIN {X 0,Y 123.675,Z 493.676,A -85,B 0,C 180,E1 -27733.138,E2 -27733.138} C_VEL
LIN {X 0,Y 123.883,Z 495.933,A -85,B 0,C 180,E1 -27736.478,E2 -27736.478} C_VEL
LIN {X 0,Y 123.805,Z 498.939,A -85,B 0,C 180,E1 -27739.913,E2 -27739.913} C_VEL
LIN {X 0,Y 123.433,Z 503.642,A -85,B 0,C 180,E1 -27744.354,E2 -27744.354} C_VEL
LIN {X 0,Y 122.748,Z 508.099,A -85,B 0,C 180,E1 -27748.001,E2 -27748.001} C_VEL
LIN {X 0,Y 121.736,Z 511.128,A -85,B 0,C 180,E1 -27750.005,E2 -27750.005} C_VEL
LIN {X 0,Y 119.702,Z 515.316,A -85,B 0,C 180,E1 -27752.475,E2 -27752.475} C_VEL
LIN {X 0,Y 118.951,Z 516.504,A -85,B 0,C 180,E1 -27753.064,E2 -27753.064} C_VEL
LIN {X 0,Y 110.131,Z 525.918,A -85,B 0,C 180,E1 -27757.089,E2 -27757.089} C_VEL
LIN {X 0,Y 101.728,Z 533.87,A -85,B 0,C 180,E1 -27762.039,E2 -27762.039} C_VEL
LIN {X 0,Y 94.15,Z 540.271,A -85,B 0,C 180,E1 -27767.791,E2 -27767.791} C_VEL
LIN {X 0,Y 86.969,Z 545.949,A -85,B 0,C 180,E1 -27775.55,E2 -27775.55} C_VEL
LIN {X 0,Y 81.426,Z 550.067,A -85,B 0,C 180,E1 -27784.433,E2 -27784.433} C_VEL
LIN {X 0,Y 78.036,Z 552.757,A -85,B 0,C 180,E1 -27794.324,E2 -27794.324} C_VEL
LIN {X 0,Y 76.65,Z 554.086,A -85,B 0,C 180,E1 -27804.739,E2 -27804.739} C_VEL
LIN {X 0,Y 76.673,Z 554.248,A -85,B 0,C 180,E1 -27809.999,E2 -27809.999} C_VEL
LIN {X 0,Y 77.113,Z 553.562,A -85,B 0,C 180,E1 -27820.502,E2 -27820.502} C_VEL
LIN {X 0,Y 79.477,Z 551.534,A -85,B 0,C 180,E1 -27830.714,E2 -27830.714} C_VEL
LIN {X 0,Y 84.016,Z 548.115,A -85,B 0,C 180,E1 -27840.126,E2 -27840.126} C_VEL
LIN {X 0,Y 90.425,Z 543.204,A -85,B 0,C 180,E1 -27848.445,E2 -27848.445} C_VEL
LIN {X 0,Y 98.361,Z 536.655,A -85,B 0,C 180,E1 -27855.603,E2 -27855.603} C_VEL
LIN {X 0,Y 106.457,Z 529.372,A -85,B 0,C 180,E1 -27860.868,E2 -27860.868} C_VEL
LIN {X 0,Y 113.993,Z 521.737,A -85,B 0,C 180,E1 -27864.775,E2 -27864.775} C_VEL
LIN {X 0,Y 118.897,Z 516.317,A -85,B 0,C 180,E1 -27866.919,E2 -27866.919} C_VEL
LIN {X 0,Y 121.19,Z 511.984,A -85,B 0,C 180,E1 -27869.367,E2 -27869.367} C_VEL
LIN {X 0,Y 122.7,Z 507.829,A -85,B 0,C 180,E1 -27872.024,E2 -27872.024} C_VEL
LIN {X 0,Y 123.326,Z 503.32,A -85,B 0,C 180,E1 -27875.754,E2 -27875.754} C_VEL
LIN {X 0,Y 123.653,Z 498.775,A -85,B 0,C 180,E1 -27880.061,E2 -27880.061} C_VEL
LIN {X 0,Y 123.702,Z 495.784,A -85,B 0,C 180,E1 -27883.497,E2 -27883.497} C_VEL
LIN {X 0,Y 123.483,Z 493.529,A -85,B 0,C 180,E1 -27886.841,E2 -27886.841} C_VEL
LIN {X 0,Y 123.319,Z 490.319,A -85,B 0,C 180,E1 -27893.455,E2 -27893.455} C_VEL
LIN {X 0,Y 123.328,Z 489.35,A -85,B 0,C 180,E1 -27896.733,E2 -27896.733} C_VEL
LIN {X 0,Y 123.336,Z 488.972,A -85,B 0,C 180,E1 -27900,E2 -27900} C_VEL
LIN {X 0,Y 123.271,Z 489.289,A -85,B 0,C 180,E1 -27903.269,E2 -27903.269} C_VEL
LIN {X 0,Y 123.115,Z 490.686,A -85,B 0,C 180,E1 -27907.646,E2 -27907.646} C_VEL
LIN {X 0,Y 123.435,Z 493.946,A -85,B 0,C 180,E1 -27914.551,E2 -27914.551} C_VEL
LIN {X 0,Y 123.834,Z 496.242,A -85,B 0,C 180,E1 -27918.189,E2 -27918.189} C_VEL
LIN {X 0,Y 123.867,Z 499.292,A -85,B 0,C 180,E1 -27921.71,E2 -27921.71} C_VEL
LIN {X 0,Y 123.467,Z 504.079,A -85,B 0,C 180,E1 -27926.177,E2 -27926.177} C_VEL
LIN {X 0,Y 122.623,Z 508.527,A -85,B 0,C 180,E1 -27929.719,E2 -27929.719} C_VEL
LIN {X 0,Y 121.088,Z 512.444,A -85,B 0,C 180,E1 -27932.249,E2 -27932.249} C_VEL
LIN {X 0,Y 120.413,Z 513.609,A -85,B 0,C 180,E1 -27932.865,E2 -27932.865} C_VEL
LIN {X 0,Y 111.861,Z 523.117,A -85,B 0,C 180,E1 -27936.769,E2 -27936.769} C_VEL
LIN {X 0,Y 103.32,Z 531.349,A -85,B 0,C 180,E1 -27941.563,E2 -27941.563} C_VEL
LIN {X 0,Y 95.202,Z 538.317,A -85,B 0,C 180,E1 -27947.58,E2 -27947.58} C_VEL
LIN {X 0,Y 89.114,Z 543.222,A -85,B 0,C 180,E1 -27953.792,E2 -27953.792} C_VEL
LIN {X 0,Y 85.946,Z 545.198,A -85,B 0,C 180,E1 -27956.81,E2 -27956.81} C_VEL
LIN {X 0,Y 79.592,Z 547.946,A -85,B 0,C 180,E1 -27961.729,E2 -27961.729} C_VEL
LIN {X 0,Y 74.814,Z 549.72,A -85,B 0,C 180,E1 -27966.252,E2 -27966.252} C_VEL
LIN {X 0,Y 72.268,Z 550.799,A -85,B 0,C 180,E1 -27970.318,E2 -27970.318} C_VEL
LIN {X 0,Y 71.754,Z 551.097,A -85,B 0,C 180,E1 -27971.806,E2 -27971.806} C_VEL
LIN {X 0,Y 70.326,Z 552.152,A -85,B 0,C 180,E1 -27978.471,E2 -27978.471} C_VEL
LIN {X 0,Y 69.647,Z 552.828,A -85,B 0,C 180,E1 -27990.001,E2 -27990.001} C_VEL
LIN {X 0,Y 70.318,Z 552.192,A -85,B 0,C 180,E1 -28001.531,E2 -28001.531} C_VEL
LIN {X 0,Y 73.147,Z 550.22,A -85,B 0,C 180,E1 -28012.602,E2 -28012.602} C_VEL
LIN {X 0,Y 78.294,Z 546.865,A -85,B 0,C 180,E1 -28022.588,E2 -28022.588} C_VEL
LIN {X 0,Y 85.372,Z 542.027,A -85,B 0,C 180,E1 -28031.192,E2 -28031.192} C_VEL
LIN {X 0,Y 91.631,Z 537.356,A -85,B 0,C 180,E1 -28036.773,E2 -28036.773} C_VEL
LIN {X 0,Y 99.962,Z 530.563,A -85,B 0,C 180,E1 -28042.275,E2 -28042.275} C_VEL
LIN {X 0,Y 109.033,Z 522.127,A -85,B 0,C 180,E1 -28046.925,E2 -28046.925} C_VEL
LIN {X 0,Y 115.444,Z 515.458,A -85,B 0,C 180,E1 -28049.591,E2 -28049.591} C_VEL
LIN {X 0,Y 116.819,Z 512.881,A -85,B 0,C 180,E1 -28051.23,E2 -28051.23} C_VEL
LIN {X 0,Y 117.825,Z 510.072,A -85,B 0,C 180,E1 -28053.473,E2 -28053.473} C_VEL
LIN {X 0,Y 118.676,Z 505.967,A -85,B 0,C 180,E1 -28057.36,E2 -28057.36} C_VEL
LIN {X 0,Y 119.076,Z 502.807,A -85,B 0,C 180,E1 -28060.794,E2 -28060.794} C_VEL
LIN {X 0,Y 119.191,Z 501.242,A -85,B 0,C 180,E1 -28062.853,E2 -28062.853} C_VEL
LIN {X 0,Y 118.968,Z 499.269,A -85,B 0,C 180,E1 -28066.332,E2 -28066.332} C_VEL
LIN {X 0,Y 118.988,Z 496.289,A -85,B 0,C 180,E1 -28073.216,E2 -28073.216} C_VEL
LIN {X 0,Y 119.228,Z 495.246,A -85,B 0,C 180,E1 -28076.62,E2 -28076.62} C_VEL
LIN {X 0,Y 119.377,Z 494.834,A -85,B 0,C 180,E1 -28080,E2 -28080} C_VEL
LIN {X 0,Y 119.293,Z 495.288,A -85,B 0,C 180,E1 -28083.377,E2 -28083.377} C_VEL
LIN {X 0,Y 119.085,Z 496.428,A -85,B 0,C 180,E1 -28086.778,E2 -28086.778} C_VEL
LIN {X 0,Y 119.121,Z 499.595,A -85,B 0,C 180,E1 -28093.65,E2 -28093.65} C_VEL
LIN {X 0,Y 119.072,Z 502.031,A -85,B 0,C 180,E1 -28097.164,E2 -28097.164} C_VEL
LIN {X 0,Y 118.289,Z 507.245,A -85,B 0,C 180,E1 -28102.717,E2 -28102.717} C_VEL
LIN {X 0,Y 117.439,Z 511.043,A -85,B 0,C 180,E1 -28106.147,E2 -28106.147} C_VEL
LIN {X 0,Y 116.32,Z 513.828,A -85,B 0,C 180,E1 -28108.216,E2 -28108.216} C_VEL
LIN {X 0,Y 114.19,Z 517.537,A -85,B 0,C 180,E1 -28110.496,E2 -28110.496} C_VEL
LIN {X 0,Y 105.983,Z 525.851,A -85,B 0,C 180,E1 -28114.012,E2 -28114.012} C_VEL
LIN {X 0,Y 97.08,Z 533.802,A -85,B 0,C 180,E1 -28118.9,E2 -28118.9} C_VEL
LIN {X 0,Y 88.993,Z 540.203,A -85,B 0,C 180,E1 -28124.703,E2 -28124.703} C_VEL
LIN {X 0,Y 81.178,Z 545.88,A -85,B 0,C 180,E1 -28132.696,E2 -28132.696} C_VEL
LIN {X 0,Y 75.052,Z 549.998,A -85,B 0,C 180,E1 -28142.081,E2 -28142.081} C_VEL
LIN {X 0,Y 71.199,Z 552.689,A -85,B 0,C 180,E1 -28152.774,E2 -28152.774} C_VEL
LIN {X 0,Y 69.573,Z 554.017,A -85,B 0,C 180,E1 -28164.202,E2 -28164.202} C_VEL
LIN {X 0,Y 69.574,Z 554.179,A -85,B 0,C 180,E1 -28169.999,E2 -28169.999} C_VEL
LIN {X 0,Y 70.111,Z 553.493,A -85,B 0,C 180,E1 -28181.565,E2 -28181.565} C_VEL
LIN {X 0,Y 72.848,Z 551.464,A -85,B 0,C 180,E1 -28192.699,E2 -28192.699} C_VEL
LIN {X 0,Y 77.931,Z 548.045,A -85,B 0,C 180,E1 -28202.758,E2 -28202.758} C_VEL
LIN {X 0,Y 84.925,Z 543.133,A -85,B 0,C 180,E1 -28211.455,E2 -28211.455} C_VEL
LIN {X 0,Y 93.503,Z 536.584,A -85,B 0,C 180,E1 -28218.732,E2 -28218.732} C_VEL
LIN {X 0,Y 102.114,Z 529.301,A -85,B 0,C 180,E1 -28223.968,E2 -28223.968} C_VEL
LIN {X 0,Y 110.048,Z 521.666,A -85,B 0,C 180,E1 -28227.799,E2 -28227.799} C_VEL
LIN {X 0,Y 114.172,Z 517.299,A -85,B 0,C 180,E1 -28229.518,E2 -28229.518} C_VEL
LIN {X 0,Y 116.241,Z 513.631,A -85,B 0,C 180,E1 -28231.781,E2 -28231.781} C_VEL
LIN {X 0,Y 117.411,Z 510.752,A -85,B 0,C 180,E1 -28233.879,E2 -28233.879} C_VEL
LIN {X 0,Y 118.145,Z 507.107,A -85,B 0,C 180,E1 -28237.253,E2 -28237.253} C_VEL
LIN {X 0,Y 118.733,Z 503.193,A -85,B 0,C 180,E1 -28241.274,E2 -28241.274} C_VEL
LIN {X 0,Y 118.951,Z 500.643,A -85,B 0,C 180,E1 -28244.491,E2 -28244.491} C_VEL
LIN {X 0,Y 118.955,Z 499.43,A -85,B 0,C 180,E1 -28246.331,E2 -28246.331} C_VEL
LIN {X 0,Y 118.966,Z 496.183,A -85,B 0,C 180,E1 -28253.215,E2 -28253.215} C_VEL
LIN {X 0,Y 119.081,Z 495.139,A -85,B 0,C 180,E1 -28256.617,E2 -28256.617} C_VEL
LIN {X 0,Y 119.14,Z 494.711,A -85,B 0,C 180,E1 -28260,E2 -28260} C_VEL
LIN {X 0,Y 119.026,Z 495.069,A -85,B 0,C 180,E1 -28263.385,E2 -28263.385} C_VEL
LIN {X 0,Y 118.755,Z 496.385,A -85,B 0,C 180,E1 -28267.564,E2 -28267.564} C_VEL
LIN {X 0,Y 118.794,Z 499.06,A -85,B 0,C 180,E1 -28273.689,E2 -28273.689} C_VEL
LIN {X 0,Y 119.023,Z 501.038,A -85,B 0,C 180,E1 -28277.172,E2 -28277.172} C_VEL
LIN {X 0,Y 118.814,Z 503.899,A -85,B 0,C 180,E1 -28280.788,E2 -28280.788} C_VEL
LIN {X 0,Y 118.213,Z 507.635,A -85,B 0,C 180,E1 -28284.593,E2 -28284.593} C_VEL
LIN {X 0,Y 117.441,Z 510.981,A -85,B 0,C 180,E1 -28287.576,E2 -28287.576} C_VEL
LIN {X 0,Y 116.107,Z 514.051,A -85,B 0,C 180,E1 -28289.807,E2 -28289.807} C_VEL
LIN {X 0,Y 115.475,Z 515.126,A -85,B 0,C 180,E1 -28290.429,E2 -28290.429} C_VEL
LIN {X 0,Y 106.417,Z 524.464,A -85,B 0,C 180,E1 -28294.358,E2 -28294.358} C_VEL
LIN {X 0,Y 97.515,Z 532.425,A -85,B 0,C 180,E1 -28299.217,E2 -28299.217} C_VEL
LIN {X 0,Y 89.466,Z 538.83,A -85,B 0,C 180,E1 -28305.01,E2 -28305.01} C_VEL
LIN {X 0,Y 81.697,Z 544.506,A -85,B 0,C 180,E1 -28312.974,E2 -28312.974} C_VEL
LIN {X 0,Y 75.421,Z 548.629,A -85,B 0,C 180,E1 -28322.231,E2 -28322.231} C_VEL
LIN {X 0,Y 71.754,Z 551.097,A -85,B 0,C 180,E1 -28331.806,E2 -28331.806} C_VEL
LIN {X 0,Y 70.039,Z 551.942,A -85,B 0,C 180,E1 -28336.323,E2 -28336.323} C_VEL
LIN {X 0,Y 67.744,Z 552.534,A -85,B 0,C 180,E1 -28340.863,E2 -28340.863} C_VEL
LIN {X 0,Y 63.494,Z 552.942,A -85,B 0,C 180,E1 -28350.695,E2 -28350.695} C_VEL
LIN {X 0,Y 62.654,Z 552.758,A -85,B 0,C 180,E1 -28356.095,E2 -28356.095} C_VEL
LIN {X 0,Y 62.71,Z 552.634,A -85,B 0,C 180,E1 -28357.92,E2 -28357.92} C_VEL
LIN {X 0,Y 64.701,Z 551.444,A -85,B 0,C 180,E1 -28369.019,E2 -28369.019} C_VEL
LIN {X 0,Y 69.171,Z 548.789,A -85,B 0,C 180,E1 -28380.532,E2 -28380.532} C_VEL
LIN {X 0,Y 76.061,Z 544.708,A -85,B 0,C 180,E1 -28390.301,E2 -28390.301} C_VEL
LIN {X 0,Y 84.53,Z 539.073,A -85,B 0,C 180,E1 -28398.442,E2 -28398.442} C_VEL
LIN {X 0,Y 93.142,Z 532.708,A -85,B 0,C 180,E1 -28404.209,E2 -28404.209} C_VEL
LIN {X 0,Y 102.543,Z 524.794,A -85,B 0,C 180,E1 -28408.951,E2 -28408.951} C_VEL
LIN {X 0,Y 110.97,Z 516.513,A -85,B 0,C 180,E1 -28412.457,E2 -28412.457} C_VEL
LIN {X 0,Y 111.973,Z 514.625,A -85,B 0,C 180,E1 -28413.937,E2 -28413.937} C_VEL
LIN {X 0,Y 113.376,Z 510.173,A -85,B 0,C 180,E1 -28418.41,E2 -28418.41} C_VEL
LIN {X 0,Y 114.016,Z 507.148,A -85,B 0,C 180,E1 -28422.049,E2 -28422.049} C_VEL
LIN {X 0,Y 114.18,Z 505.907,A -85,B 0,C 180,E1 -28423.919,E2 -28423.919} C_VEL
LIN {X 0,Y 114.122,Z 502.99,A -85,B 0,C 180,E1 -28430.178,E2 -28430.178} C_VEL
LIN {X 0,Y 114.687,Z 500.835,A -85,B 0,C 180,E1 -28436.486,E2 -28436.486} C_VEL
LIN {X 0,Y 114.913,Z 500.363,A -85,B 0,C 180,E1 -28440,E2 -28440} C_VEL
LIN {X 0,Y 114.734,Z 500.908,A -85,B 0,C 180,E1 -28443.512,E2 -28443.512} C_VEL
LIN {X 0,Y 114.28,Z 503.359,A -85,B 0,C 180,E1 -28450.27,E2 -28450.27} C_VEL
LIN {X 0,Y 114.202,Z 505.386,A -85,B 0,C 180,E1 -28454.25,E2 -28454.25} C_VEL
LIN {X 0,Y 114.078,Z 506.606,A -85,B 0,C 180,E1 -28456.095,E2 -28456.095} C_VEL
LIN {X 0,Y 113.057,Z 510.941,A -85,B 0,C 180,E1 -28461.178,E2 -28461.178} C_VEL
LIN {X 0,Y 112.184,Z 513.774,A -85,B 0,C 180,E1 -28464.029,E2 -28464.029} C_VEL
LIN {X 0,Y 110.943,Z 516.57,A -85,B 0,C 180,E1 -28466.323,E2 -28466.323} C_VEL
LIN {X 0,Y 109.294,Z 518.958,A -85,B 0,C 180,E1 -28467.849,E2 -28467.849} C_VEL
LIN {X 0,Y 100.784,Z 527.017,A -85,B 0,C 180,E1 -28471.324,E2 -28471.324} C_VEL
LIN {X 0,Y 91.489,Z 534.744,A -85,B 0,C 180,E1 -28476.235,E2 -28476.235} C_VEL
LIN {X 0,Y 84.128,Z 540.135,A -85,B 0,C 180,E1 -28481.248,E2 -28481.248} C_VEL
LIN {X 0,Y 77.612,Z 544.567,A -85,B 0,C 180,E1 -28487.222,E2 -28487.222} C_VEL
LIN {X 0,Y 72.03,Z 548.057,A -85,B 0,C 180,E1 -28494.166,E2 -28494.166} C_VEL
LIN {X 0,Y 66.306,Z 551.447,A -85,B 0,C 180,E1 -28504.914,E2 -28504.914} C_VEL
LIN {X 0,Y 63.152,Z 553.452,A -85,B 0,C 180,E1 -28517.139,E2 -28517.139} C_VEL
LIN {X 0,Y 62.492,Z 554.111,A -85,B 0,C 180,E1 -28529.999,E2 -28529.999} C_VEL
LIN {X 0,Y 63.152,Z 553.423,A -85,B 0,C 180,E1 -28542.86,E2 -28542.86} C_VEL
LIN {X 0,Y 66.305,Z 551.394,A -85,B 0,C 180,E1 -28555.086,E2 -28555.086} C_VEL
LIN {X 0,Y 72.038,Z 547.975,A -85,B 0,C 180,E1 -28565.828,E2 -28565.828} C_VEL
LIN {X 0,Y 79.698,Z 543.062,A -85,B 0,C 180,E1 -28574.866,E2 -28574.866} C_VEL
LIN {X 0,Y 88.95,Z 536.514,A -85,B 0,C 180,E1 -28582.195,E2 -28582.195} C_VEL
LIN {X 0,Y 98.09,Z 529.23,A -85,B 0,C 180,E1 -28587.338,E2 -28587.338} C_VEL
LIN {X 0,Y 106.431,Z 521.595,A -85,B 0,C 180,E1 -28591.038,E2 -28591.038} C_VEL
LIN {X 0,Y 109.287,Z 518.715,A -85,B 0,C 180,E1 -28592.157,E2 -28592.157} C_VEL
LIN {X 0,Y 110.844,Z 516.417,A -85,B 0,C 180,E1 -28593.652,E2 -28593.652} C_VEL
LIN {X 0,Y 111.69,Z 514.768,A -85,B 0,C 180,E1 -28594.866,E2 -28594.866} C_VEL
LIN {X 0,Y 112.735,Z 511.526,A -85,B 0,C 180,E1 -28598.035,E2 -28598.035} C_VEL
LIN {X 0,Y 113.584,Z 507.958,A -85,B 0,C 180,E1 -28601.979,E2 -28601.979} C_VEL
LIN {X 0,Y 113.93,Z 506.447,A -85,B 0,C 180,E1 -28603.884,E2 -28603.884} C_VEL
LIN {X 0,Y 114.042,Z 505.228,A -85,B 0,C 180,E1 -28605.729,E2 -28605.729} C_VEL
LIN {X 0,Y 114.157,Z 503.006,A -85,B 0,C 180,E1 -28610.072,E2 -28610.072} C_VEL
LIN {X 0,Y 114.324,Z 501.828,A -85,B 0,C 180,E1 -28612.938,E2 -28612.938} C_VEL
LIN {X 0,Y 114.557,Z 500.729,A -85,B 0,C 180,E1 -28616.483,E2 -28616.483} C_VEL
LIN {X 0,Y 114.674,Z 500.253,A -85,B 0,C 180,E1 -28620,E2 -28620} C_VEL
LIN {X 0,Y 114.499,Z 500.658,A -85,B 0,C 180,E1 -28623.519,E2 -28623.519} C_VEL
LIN {X 0,Y 113.995,Z 502.617,A -85,B 0,C 180,E1 -28629.452,E2 -28629.452} C_VEL
LIN {X 0,Y 114.025,Z 505.7,A -85,B 0,C 180,E1 -28636.103,E2 -28636.103} C_VEL
LIN {X 0,Y 113.914,Z 506.897,A -85,B 0,C 180,E1 -28637.968,E2 -28637.968} C_VEL
LIN {X 0,Y 113.225,Z 510.149,A -85,B 0,C 180,E1 -28641.866,E2 -28641.866} C_VEL
LIN {X 0,Y 112.342,Z 513.147,A -85,B 0,C 180,E1 -28644.978,E2 -28644.978} C_VEL
LIN {X 0,Y 111.937,Z 514.322,A -85,B 0,C 180,E1 -28646.072,E2 -28646.072} C_VEL
LIN {X 0,Y 110.975,Z 516.203,A -85,B 0,C 180,E1 -28647.549,E2 -28647.549} C_VEL
LIN {X 0,Y 102.571,Z 524.535,A -85,B 0,C 180,E1 -28651.077,E2 -28651.077} C_VEL
LIN {X 0,Y 93.182,Z 532.496,A -85,B 0,C 180,E1 -28655.827,E2 -28655.827} C_VEL
LIN {X 0,Y 84.233,Z 539.143,A -85,B 0,C 180,E1 -28661.874,E2 -28661.874} C_VEL
LIN {X 0,Y 76.115,Z 544.576,A -85,B 0,C 180,E1 -28669.735,E2 -28669.735} C_VEL
LIN {X 0,Y 69.189,Z 548.699,A -85,B 0,C 180,E1 -28679.477,E2 -28679.477} C_VEL
LIN {X 0,Y 64.723,Z 551.386,A -85,B 0,C 180,E1 -28690.989,E2 -28690.989} C_VEL
LIN {X 0,Y 62.607,Z 552.725,A -85,B 0,C 180,E1 -28703.555,E2 -28703.555} C_VEL
LIN {X 0,Y 62.548,Z 552.897,A -85,B 0,C 180,E1 -28710.001,E2 -28710.001} C_VEL
LIN {X 0,Y 62.71,Z 552.634,A -85,B 0,C 180,E1 -28717.92,E2 -28717.92} C_VEL
LIN {X 0,Y 62.707,Z 552.227,A -85,B 0,C 180,E1 -28723.305,E2 -28723.305} C_VEL
LIN {X 0,Y 61.931,Z 551.085,A -85,B 0,C 180,E1 -28732.364,E2 -28732.364} C_VEL
LIN {X 0,Y 62.198,Z 549.803,A -85,B 0,C 180,E1 -28739.64,E2 -28739.64} C_VEL
LIN {X 0,Y 63.767,Z 548.558,A -85,B 0,C 180,E1 -28744.724,E2 -28744.724} C_VEL
LIN {X 0,Y 64.638,Z 548.045,A -85,B 0,C 180,E1 -28746.249,E2 -28746.249} C_VEL
LIN {X 0,Y 70.758,Z 544.776,A -85,B 0,C 180,E1 -28754.05,E2 -28754.05} C_VEL
LIN {X 0,Y 78.77,Z 539.935,A -85,B 0,C 180,E1 -28761.35,E2 -28761.35} C_VEL
LIN {X 0,Y 87.798,Z 533.781,A -85,B 0,C 180,E1 -28767.193,E2 -28767.193} C_VEL
LIN {X 0,Y 97.603,Z 526.089,A -85,B 0,C 180,E1 -28771.895,E2 -28771.895} C_VEL
LIN {X 0,Y 104.931,Z 519.542,A -85,B 0,C 180,E1 -28774.716,E2 -28774.716} C_VEL
LIN {X 0,Y 106.268,Z 518.094,A -85,B 0,C 180,E1 -28775.371,E2 -28775.371} C_VEL
LIN {X 0,Y 107.012,Z 516.6,A -85,B 0,C 180,E1 -28776.846,E2 -28776.846} C_VEL
LIN {X 0,Y 108.345,Z 512.996,A -85,B 0,C 180,E1 -28781.074,E2 -28781.074} C_VEL
LIN {X 0,Y 108.814,Z 511.521,A -85,B 0,C 180,E1 -28783.103,E2 -28783.103} C_VEL
LIN {X 0,Y 109.034,Z 510.302,A -85,B 0,C 180,E1 -28785.208,E2 -28785.208} C_VEL
LIN {X 0,Y 109.387,Z 507.329,A -85,B 0,C 180,E1 -28792.617,E2 -28792.617} C_VEL
LIN {X 0,Y 109.851,Z 506.226,A -85,B 0,C 180,E1 -28796.332,E2 -28796.332} C_VEL
LIN {X 0,Y 110.175,Z 505.694,A -85,B 0,C 180,E1 -28800,E2 -28800} C_VEL
LIN {X 0,Y 109.902,Z 506.303,A -85,B 0,C 180,E1 -28803.666,E2 -28803.666} C_VEL
LIN {X 0,Y 109.507,Z 507.468,A -85,B 0,C 180,E1 -28807.374,E2 -28807.374} C_VEL
LIN {X 0,Y 109.196,Z 509.014,A -85,B 0,C 180,E1 -28811.133,E2 -28811.133} C_VEL
LIN {X 0,Y 108.945,Z 510.99,A -85,B 0,C 180,E1 -28814.953,E2 -28814.953} C_VEL
LIN {X 0,Y 107.899,Z 514.088,A -85,B 0,C 180,E1 -28819.006,E2 -28819.006} C_VEL
LIN {X 0,Y 106.621,Z 517.379,A -85,B 0,C 180,E1 -28822.657,E2 -28822.657} C_VEL
LIN {X 0,Y 105.39,Z 519.479,A -85,B 0,C 180,E1 -28824.453,E2 -28824.453} C_VEL
LIN {X 0,Y 104.486,Z 520.544,A -85,B 0,C 180,E1 -28825.03,E2 -28825.03} C_VEL
LIN {X 0,Y 95.826,Z 528.182,A -85,B 0,C 180,E1 -28828.345,E2 -28828.345} C_VEL
LIN {X 0,Y 87.447,Z 534.676,A -85,B 0,C 180,E1 -28832.448,E2 -28832.448} C_VEL
LIN {X 0,Y 79.602,Z 540.067,A -85,B 0,C 180,E1 -28837.381,E2 -28837.381} C_VEL
LIN {X 0,Y 72.513,Z 544.499,A -85,B 0,C 180,E1 -28843.372,E2 -28843.372} C_VEL
LIN {X 0,Y 66.376,Z 547.988,A -85,B 0,C 180,E1 -28850.558,E2 -28850.558} C_VEL
LIN {X 0,Y 59.906,Z 551.379,A -85,B 0,C 180,E1 -28862.012,E2 -28862.012} C_VEL
LIN {X 0,Y 56.244,Z 553.384,A -85,B 0,C 180,E1 -28875.527,E2 -28875.527} C_VEL
LIN {X 0,Y 55.393,Z 554.042,A -85,B 0,C 180,E1 -28889.999,E2 -28889.999} C_VEL
LIN {X 0,Y 56.244,Z 553.354,A -85,B 0,C 180,E1 -28904.472,E2 -28904.472} C_VEL
LIN {X 0,Y 59.905,Z 551.324,A -85,B 0,C 180,E1 -28917.987,E2 -28917.987} C_VEL
LIN {X 0,Y 66.386,Z 547.905,A -85,B 0,C 180,E1 -28929.434,E2 -28929.434} C_VEL
LIN {X 0,Y 74.793,Z 542.992,A -85,B 0,C 180,E1 -28938.74,E2 -28938.74} C_VEL
LIN {X 0,Y 84.768,Z 536.443,A -85,B 0,C 180,E1 -28946.005,E2 -28946.005} C_VEL
LIN {X 0,Y 94.417,Z 529.159,A -85,B 0,C 180,E1 -28950.999,E2 -28950.999} C_VEL
LIN {X 0,Y 104.433,Z 520.357,A -85,B 0,C 180,E1 -28954.947,E2 -28954.947} C_VEL
LIN {X 0,Y 105.335,Z 519.264,A -85,B 0,C 180,E1 -28955.56,E2 -28955.56} C_VEL
LIN {X 0,Y 106.607,Z 517.129,A -85,B 0,C 180,E1 -28957.359,E2 -28957.359} C_VEL
LIN {X 0,Y 107.783,Z 513.923,A -85,B 0,C 180,E1 -28960.973,E2 -28960.973} C_VEL
LIN {X 0,Y 108.858,Z 510.504,A -85,B 0,C 180,E1 -28965.561,E2 -28965.561} C_VEL
LIN {X 0,Y 109.079,Z 508.819,A -85,B 0,C 180,E1 -28968.855,E2 -28968.855} C_VEL
LIN {X 0,Y 109.394,Z 507.262,A -85,B 0,C 180,E1 -28972.618,E2 -28972.618} C_VEL
LIN {X 0,Y 109.743,Z 506.128,A -85,B 0,C 180,E1 -28976.329,E2 -28976.329} C_VEL
LIN {X 0,Y 109.948,Z 505.582,A -85,B 0,C 180,E1 -28980,E2 -28980} C_VEL
LIN {X 0,Y 109.678,Z 506.056,A -85,B 0,C 180,E1 -28983.674,E2 -28983.674} C_VEL
LIN {X 0,Y 109.252,Z 507.124,A -85,B 0,C 180,E1 -28987.392,E2 -28987.392} C_VEL
LIN {X 0,Y 108.882,Z 510.179,A -85,B 0,C 180,E1 -28994.963,E2 -28994.963} C_VEL
LIN {X 0,Y 108.72,Z 511.285,A -85,B 0,C 180,E1 -28996.912,E2 -28996.912} C_VEL
LIN {X 0,Y 107.621,Z 514.68,A -85,B 0,C 180,E1 -29001.301,E2 -29001.301} C_VEL
LIN {X 0,Y 106.239,Z 517.823,A -85,B 0,C 180,E1 -29004.65,E2 -29004.65} C_VEL
LIN {X 0,Y 103.461,Z 520.629,A -85,B 0,C 180,E1 -29005.835,E2 -29005.835} C_VEL
LIN {X 0,Y 93.362,Z 529.354,A -85,B 0,C 180,E1 -29010.04,E2 -29010.04} C_VEL
LIN {X 0,Y 85.152,Z 535.498,A -85,B 0,C 180,E1 -29014.377,E2 -29014.377} C_VEL
LIN {X 0,Y 77.862,Z 540.396,A -85,B 0,C 180,E1 -29019.436,E2 -29019.436} C_VEL
LIN {X 0,Y 70.805,Z 544.647,A -85,B 0,C 180,E1 -29025.989,E2 -29025.989} C_VEL
LIN {X 0,Y 63.149,Z 548.769,A -85,B 0,C 180,E1 -29036.189,E2 -29036.189} C_VEL
LIN {X 0,Y 58.023,Z 551.456,A -85,B 0,C 180,E1 -29048.693,E2 -29048.693} C_VEL
LIN {X 0,Y 55.564,Z 552.794,A -85,B 0,C 180,E1 -29062.734,E2 -29062.734} C_VEL
LIN {X 0,Y 55.466,Z 552.966,A -85,B 0,C 180,E1 -29070.001,E2 -29070.001} C_VEL
LIN {X 0,Y 56.452,Z 552.329,A -85,B 0,C 180,E1 -29084.418,E2 -29084.418} C_VEL
